LIN {X 0,Y 186.406,Z 165.264,A -85,B 0,C 180,E1 -22320.001,E2 -22320.001} C_VEL
LIN {X 0,Y 185.926,Z 165.321,A -85,B 0,C 180,E1 -22324.336,E2 -22324.336} C_VEL
LIN {X 0,Y 186.028,Z 165.314,A -85,B 0,C 180,E1 -22328.692,E2 -22328.692} C_VEL
LIN {X 0,Y 185.764,Z 165.342,A -85,B 0,C 180,E1 -22333.121,E2 -22333.121} C_VEL
LIN {X 0,Y 185.673,Z 165.354,A -85,B 0,C 180,E1 -22338.867,E2 -22338.867} C_VEL
LIN {X 0,Y 185.576,Z 165.369,A -85,B 0,C 180,E1 -22344.647,E2 -22344.647} C_VEL
LIN {X 0,Y 185.579,Z 165.363,A -85,B 0,C 180,E1 -22349.494,E2 -22349.494} C_VEL
LIN {X 0,Y 185.519,Z 165.374,A -85,B 0,C 180,E1 -22354.629,E2 -22354.629} C_VEL
LIN {X 0,Y 185.544,Z 165.367,A -85,B 0,C 180,E1 -22357.305,E2 -22357.305} C_VEL
LIN {X 0,Y 185.504,Z 165.377,A -85,B 0,C 180,E1 -22360.738,E2 -22360.738} C_VEL
LIN {X 0,Y 185.508,Z 165.375,A -85,B 0,C 180,E1 -22363.962,E2 -22363.962} C_VEL
LIN {X 0,Y 185.485,Z 165.38,A -85,B 0,C 180,E1 -22369.272,E2 -22369.272} C_VEL
LIN {X 0,Y 185.627,Z 165.502,A -85,B 0,C 180,E1 -22372.033,E2 -22372.033} C_VEL
LIN {X 0,Y 187.759,Z 175.884,A -85,B 0,C 180,E1 -22376.802,E2 -22376.802} C_VEL
LIN {X 0,Y 192.861,Z 193.887,A -85,B 0,C 180,E1 -22378.301,E2 -22378.301} C_VEL
LIN {X 0,Y 196.312,Z 235.606,A -85,B 0,C 180,E1 -22380.852,E2 -22380.852} C_VEL
LIN {X 0,Y 194.6,Z 269.087,A -85,B 0,C 180,E1 -22382.53,E2 -22382.53} C_VEL
LIN {X 0,Y 193.581,Z 274.86,A -85,B 0,C 180,E1 -22382.768,E2 -22382.768} C_VEL
LIN {X 0,Y 190.128,Z 284.123,A -85,B 0,C 180,E1 -22383.093,E2 -22383.093} C_VEL
LIN {X 0,Y 186.695,Z 293.281,A -85,B 0,C 180,E1 -22383.622,E2 -22383.622} C_VEL
LIN {X 0,Y 185.665,Z 298.885,A -85,B 0,C 180,E1 -22384.126,E2 -22384.126} C_VEL
LIN {X 0,Y 184.294,Z 310.636,A -85,B 0,C 180,E1 -22385.5,E2 -22385.5} C_VEL
LIN {X 0,Y 182.538,Z 323.588,A -85,B 0,C 180,E1 -22387.526,E2 -22387.526} C_VEL
LIN {X 0,Y 180.854,Z 335.007,A -85,B 0,C 180,E1 -22389.826,E2 -22389.826} C_VEL
LIN {X 0,Y 179.322,Z 344.82,A -85,B 0,C 180,E1 -22392.319,E2 -22392.319} C_VEL
LIN {X 0,Y 178.255,Z 353.885,A -85,B 0,C 180,E1 -22395.152,E2 -22395.152} C_VEL
LIN {X 0,Y 177.417,Z 361.323,A -85,B 0,C 180,E1 -22397.998,E2 -22397.998} C_VEL
LIN {X 0,Y 176.901,Z 368.603,A -85,B 0,C 180,E1 -22401.433,E2 -22401.433} C_VEL
LIN {X 0,Y 176.798,Z 373.802,A -85,B 0,C 180,E1 -22404.512,E2 -22404.512} C_VEL
LIN {X 0,Y 176.75,Z 378.056,A -85,B 0,C 180,E1 -22407.722,E2 -22407.722} C_VEL
LIN {X 0,Y 176.865,Z 380.423,A -85,B 0,C 180,E1 -22410.001,E2 -22410.001} C_VEL
LIN {X 0,Y 176.496,Z 382.213,A -85,B 0,C 180,E1 -22412.283,E2 -22412.283} C_VEL
LIN {X 0,Y 176.293,Z 383.654,A -85,B 0,C 180,E1 -22414.69,E2 -22414.69} C_VEL
LIN {X 0,Y 176.459,Z 385.146,A -85,B 0,C 180,E1 -22419.168,E2 -22419.168} C_VEL
LIN {X 0,Y 177.62,Z 385.137,A -85,B 0,C 180,E1 -22423.734,E2 -22423.734} C_VEL
LIN {X 0,Y 180.063,Z 383.679,A -85,B 0,C 180,E1 -22428.195,E2 -22428.195} C_VEL
LIN {X 0,Y 181.747,Z 382.388,A -85,B 0,C 180,E1 -22430.367,E2 -22430.367} C_VEL
LIN {X 0,Y 185.887,Z 378.597,A -85,B 0,C 180,E1 -22434.576,E2 -22434.576} C_VEL
LIN {X 0,Y 189.751,Z 374.715,A -85,B 0,C 180,E1 -22437.58,E2 -22437.58} C_VEL
LIN {X 0,Y 194.332,Z 369.791,A -85,B 0,C 180,E1 -22440.419,E2 -22440.419} C_VEL
LIN {X 0,Y 200.257,Z 362.613,A -85,B 0,C 180,E1 -22443.556,E2 -22443.556} C_VEL
LIN {X 0,Y 206.088,Z 355.024,A -85,B 0,C 180,E1 -22446.034,E2 -22446.034} C_VEL
LIN {X 0,Y 212.388,Z 345.713,A -85,B 0,C 180,E1 -22448.349,E2 -22448.349} C_VEL
LIN {X 0,Y 219.022,Z 334.32,A -85,B 0,C 180,E1 -22450.526,E2 -22450.526} C_VEL
LIN {X 0,Y 224.449,Z 323.763,A -85,B 0,C 180,E1 -22452.014,E2 -22452.014} C_VEL
LIN {X 0,Y 230.105,Z 310.634,A -85,B 0,C 180,E1 -22453.41,E2 -22453.41} C_VEL
LIN {X 0,Y 234.374,Z 298.405,A -85,B 0,C 180,E1 -22454.352,E2 -22454.352} C_VEL
LIN {X 0,Y 238.04,Z 284.522,A -85,B 0,C 180,E1 -22455.167,E2 -22455.167} C_VEL
LIN {X 0,Y 241.045,Z 267.551,A -85,B 0,C 180,E1 -22455.878,E2 -22455.878} C_VEL
LIN {X 0,Y 243.195,Z 253.201,A -85,B 0,C 180,E1 -22456.447,E2 -22456.447} C_VEL
LIN {X 0,Y 241.769,Z 247.758,A -85,B 0,C 180,E1 -22458.324,E2 -22458.324} C_VEL
LIN {X 0,Y 240.721,Z 244.112,A -85,B 0,C 180,E1 -22459.965,E2 -22459.965} C_VEL
LIN {X 0,Y 239.6,Z 240.401,A -85,B 0,C 180,E1 -22462.093,E2 -22462.093} C_VEL
LIN {X 0,Y 238.583,Z 236.055,A -85,B 0,C 180,E1 -22466.094,E2 -22466.094} C_VEL
LIN {X 0,Y 238.441,Z 235.364,A -85,B 0,C 180,E1 -22467.957,E2 -22467.957} C_VEL
LIN {X 0,Y 238.94,Z 235.62,A -85,B 0,C 180,E1 -22471.095,E2 -22471.095} C_VEL
LIN {X 0,Y 240.37,Z 237.492,A -85,B 0,C 180,E1 -22474.306,E2 -22474.306} C_VEL
LIN {X 0,Y 241.967,Z 240.386,A -85,B 0,C 180,E1 -22476.642,E2 -22476.642} C_VEL
LIN {X 0,Y 243.416,Z 243.368,A -85,B 0,C 180,E1 -22478.363,E2 -22478.363} C_VEL
LIN {X 0,Y 244.149,Z 244.907,A -85,B 0,C 180,E1 -22479.131,E2 -22479.131} C_VEL
LIN {X 0,Y 239.788,Z 272.332,A -85,B 0,C 180,E1 -22480.254,E2 -22480.254} C_VEL
LIN {X 0,Y 236.802,Z 285.281,A -85,B 0,C 180,E1 -22481.057,E2 -22481.057} C_VEL
LIN {X 0,Y 232.723,Z 298.537,A -85,B 0,C 180,E1 -22482.195,E2 -22482.195} C_VEL
LIN {X 0,Y 228.104,Z 310.509,A -85,B 0,C 180,E1 -22483.583,E2 -22483.583} C_VEL
LIN {X 0,Y 223.03,Z 321.088,A -85,B 0,C 180,E1 -22485.141,E2 -22485.141} C_VEL
LIN {X 0,Y 217.786,Z 330.518,A -85,B 0,C 180,E1 -22486.944,E2 -22486.944} C_VEL
LIN {X 0,Y 212.304,Z 339.171,A -85,B 0,C 180,E1 -22489.026,E2 -22489.026} C_VEL
LIN {X 0,Y 207.525,Z 345.733,A -85,B 0,C 180,E1 -22491.023,E2 -22491.023} C_VEL
LIN {X 0,Y 202.253,Z 352.165,A -85,B 0,C 180,E1 -22493.515,E2 -22493.515} C_VEL
LIN {X 0,Y 197.206,Z 357.616,A -85,B 0,C 180,E1 -22496.261,E2 -22496.261} C_VEL
LIN {X 0,Y 192.887,Z 361.653,A -85,B 0,C 180,E1 -22498.955,E2 -22498.955} C_VEL
LIN {X 0,Y 188.616,Z 365.071,A -85,B 0,C 180,E1 -22502.135,E2 -22502.135} C_VEL
LIN {X 0,Y 186.132,Z 366.712,A -85,B 0,C 180,E1 -22504.33,E2 -22504.33} C_VEL
LIN {X 0,Y 183.894,Z 367.917,A -85,B 0,C 180,E1 -22506.583,E2 -22506.583} C_VEL
LIN {X 0,Y 182.006,Z 368.679,A -85,B 0,C 180,E1 -22508.884,E2 -22508.884} C_VEL
LIN {X 0,Y 179.738,Z 368.959,A -85,B 0,C 180,E1 -22512.164,E2 -22512.164} C_VEL
LIN {X 0,Y 177.81,Z 368.208,A -85,B 0,C 180,E1 -22516.061,E2 -22516.061} C_VEL
LIN {X 0,Y 176.957,Z 367.125,A -85,B 0,C 180,E1 -22518.525,E2 -22518.525} C_VEL
LIN {X 0,Y 176.371,Z 365.541,A -85,B 0,C 180,E1 -22521.015,E2 -22521.015} C_VEL
LIN {X 0,Y 176.006,Z 362.223,A -85,B 0,C 180,E1 -22524.788,E2 -22524.788} C_VEL
LIN {X 0,Y 176.163,Z 357.578,A -85,B 0,C 180,E1 -22528.634,E2 -22528.634} C_VEL
LIN {X 0,Y 176.704,Z 351.736,A -85,B 0,C 180,E1 -22532.314,E2 -22532.314} C_VEL
LIN {X 0,Y 177.477,Z 344.811,A -85,B 0,C 180,E1 -22535.738,E2 -22535.738} C_VEL
LIN {X 0,Y 178.528,Z 336.49,A -85,B 0,C 180,E1 -22539.039,E2 -22539.039} C_VEL
LIN {X 0,Y 179.917,Z 326.961,A -85,B 0,C 180,E1 -22542.081,E2 -22542.081} C_VEL
LIN {X 0,Y 181.44,Z 315.862,A -85,B 0,C 180,E1 -22544.909,E2 -22544.909} C_VEL
LIN {X 0,Y 183.087,Z 304.373,A -85,B 0,C 180,E1 -22547.233,E2 -22547.233} C_VEL
LIN {X 0,Y 184.588,Z 292.093,A -85,B 0,C 180,E1 -22549.175,E2 -22549.175} C_VEL
LIN {X 0,Y 185.917,Z 279.648,A -85,B 0,C 180,E1 -22550.683,E2 -22550.683} C_VEL
LIN {X 0,Y 186.97,Z 265.297,A -85,B 0,C 180,E1 -22551.917,E2 -22551.917} C_VEL
LIN {X 0,Y 190.086,Z 210.466,A -85,B 0,C 180,E1 -22554.824,E2 -22554.824} C_VEL
LIN {X 0,Y 190.673,Z 200.076,A -85,B 0,C 180,E1 -22555.357,E2 -22555.357} C_VEL
LIN {X 0,Y 179.22,Z 168.469,A -85,B 0,C 180,E1 -22558.282,E2 -22558.282} C_VEL
LIN {X 0,Y 178.56,Z 166.317,A -85,B 0,C 180,E1 -22558.483,E2 -22558.483} C_VEL
LIN {X 0,Y 178.513,Z 166.249,A -85,B 0,C 180,E1 -22564.337,E2 -22564.337} C_VEL
LIN {X 0,Y 178.521,Z 166.249,A -85,B 0,C 180,E1 -22569.248,E2 -22569.248} C_VEL
LIN {X 0,Y 178.614,Z 166.236,A -85,B 0,C 180,E1 -22571.652,E2 -22571.652} C_VEL
LIN {X 0,Y 178.649,Z 166.226,A -85,B 0,C 180,E1 -22576.346,E2 -22576.346} C_VEL
LIN {X 0,Y 178.958,Z 166.195,A -85,B 0,C 180,E1 -22580.961,E2 -22580.961} C_VEL
LIN {X 0,Y 179.153,Z 166.167,A -85,B 0,C 180,E1 -22587.751,E2 -22587.751} C_VEL
LIN {X 0,Y 179.369,Z 166.141,A -85,B 0,C 180,E1 -22589.999,E2 -22589.999} C_VEL
LIN {X 0,Y 178.872,Z 166.201,A -85,B 0,C 180,E1 -22594.506,E2 -22594.506} C_VEL
LIN {X 0,Y 178.958,Z 166.191,A -85,B 0,C 180,E1 -22599.037,E2 -22599.037} C_VEL
LIN {X 0,Y 178.679,Z 166.226,A -85,B 0,C 180,E1 -22603.65,E2 -22603.65} C_VEL
LIN {X 0,Y 178.62,Z 166.23,A -85,B 0,C 180,E1 -22609.215,E2 -22609.215} C_VEL
LIN {X 0,Y 178.517,Z 166.246,A -85,B 0,C 180,E1 -22615.114,E2 -22615.114} C_VEL
LIN {X 0,Y 178.52,Z 166.246,A -85,B 0,C 180,E1 -22619.993,E2 -22619.993} C_VEL
LIN {X 0,Y 178.482,Z 166.251,A -85,B 0,C 180,E1 -22624.219,E2 -22624.219} C_VEL
LIN {X 0,Y 178.47,Z 166.252,A -85,B 0,C 180,E1 -22629.054,E2 -22629.054} C_VEL
LIN {X 0,Y 178.497,Z 166.25,A -85,B 0,C 180,E1 -22632.015,E2 -22632.015} C_VEL
LIN {X 0,Y 178.514,Z 166.243,A -85,B 0,C 180,E1 -22635.124,E2 -22635.124} C_VEL
LIN {X 0,Y 178.498,Z 166.25,A -85,B 0,C 180,E1 -22638.424,E2 -22638.424} C_VEL
LIN {X 0,Y 178.456,Z 166.254,A -85,B 0,C 180,E1 -22643.792,E2 -22643.792} C_VEL
LIN {X 0,Y 178.489,Z 166.25,A -85,B 0,C 180,E1 -22646.548,E2 -22646.548} C_VEL
LIN {X 0,Y 178.52,Z 166.243,A -85,B 0,C 180,E1 -22650.007,E2 -22650.007} C_VEL
LIN {X 0,Y 178.532,Z 166.246,A -85,B 0,C 180,E1 -22654.876,E2 -22654.876} C_VEL
LIN {X 0,Y 178.621,Z 166.232,A -85,B 0,C 180,E1 -22660.784,E2 -22660.784} C_VEL
LIN {X 0,Y 178.663,Z 166.229,A -85,B 0,C 180,E1 -22664.018,E2 -22664.018} C_VEL
LIN {X 0,Y 178.859,Z 166.204,A -85,B 0,C 180,E1 -22669.211,E2 -22669.211} C_VEL
LIN {X 0,Y 178.923,Z 166.197,A -85,B 0,C 180,E1 -22673.233,E2 -22673.233} C_VEL
LIN {X 0,Y 179.152,Z 166.167,A -85,B 0,C 180,E1 -22677.753,E2 -22677.753} C_VEL
LIN {X 0,Y 179.369,Z 166.141,A -85,B 0,C 180,E1 -22680.001,E2 -22680.001} C_VEL
LIN {X 0,Y 178.875,Z 166.199,A -85,B 0,C 180,E1 -22684.508,E2 -22684.508} C_VEL
LIN {X 0,Y 178.977,Z 166.19,A -85,B 0,C 180,E1 -22689.038,E2 -22689.038} C_VEL
LIN {X 0,Y 178.681,Z 166.224,A -85,B 0,C 180,E1 -22693.651,E2 -22693.651} C_VEL
LIN {X 0,Y 178.621,Z 166.231,A -85,B 0,C 180,E1 -22699.216,E2 -22699.216} C_VEL
LIN {X 0,Y 178.519,Z 166.247,A -85,B 0,C 180,E1 -22705.115,E2 -22705.115} C_VEL
LIN {X 0,Y 178.523,Z 166.244,A -85,B 0,C 180,E1 -22709.995,E2 -22709.995} C_VEL
LIN {X 0,Y 178.496,Z 166.251,A -85,B 0,C 180,E1 -22714.226,E2 -22714.226} C_VEL
LIN {X 0,Y 178.426,Z 166.257,A -85,B 0,C 180,E1 -22719.067,E2 -22719.067} C_VEL
LIN {X 0,Y 178.43,Z 166.26,A -85,B 0,C 180,E1 -22722.037,E2 -22722.037} C_VEL
LIN {X 0,Y 178.422,Z 166.255,A -85,B 0,C 180,E1 -22725.156,E2 -22725.156} C_VEL
LIN {X 0,Y 178.541,Z 166.245,A -85,B 0,C 180,E1 -22731.398,E2 -22731.398} C_VEL
LIN {X 0,Y 178.565,Z 166.455,A -85,B 0,C 180,E1 -22731.709,E2 -22731.709} C_VEL
LIN {X 0,Y 180.436,Z 175.467,A -85,B 0,C 180,E1 -22736.027,E2 -22736.027} C_VEL
LIN {X 0,Y 186.131,Z 195.279,A -85,B 0,C 180,E1 -22737.754,E2 -22737.754} C_VEL
LIN {X 0,Y 189.408,Z 236.226,A -85,B 0,C 180,E1 -22740.353,E2 -22740.353} C_VEL
LIN {X 0,Y 186.805,Z 285.736,A -85,B 0,C 180,E1 -22743.012,E2 -22743.012} C_VEL
LIN {X 0,Y 185.665,Z 298.885,A -85,B 0,C 180,E1 -22744.126,E2 -22744.126} C_VEL
LIN {X 0,Y 184.474,Z 304.383,A -85,B 0,C 180,E1 -22744.679,E2 -22744.679} C_VEL
LIN {X 0,Y 180.587,Z 312.949,A -85,B 0,C 180,E1 -22745.665,E2 -22745.665} C_VEL
LIN {X 0,Y 176.518,Z 321.185,A -85,B 0,C 180,E1 -22746.903,E2 -22746.903} C_VEL
LIN {X 0,Y 175.066,Z 326.174,A -85,B 0,C 180,E1 -22747.839,E2 -22747.839} C_VEL
LIN {X 0,Y 173.279,Z 337.827,A -85,B 0,C 180,E1 -22750.452,E2 -22750.452} C_VEL
LIN {X 0,Y 171.811,Z 348.066,A -85,B 0,C 180,E1 -22753.362,E2 -22753.362} C_VEL
LIN {X 0,Y 170.824,Z 356.454,A -85,B 0,C 180,E1 -22756.317,E2 -22756.317} C_VEL
LIN {X 0,Y 170.017,Z 364.622,A -85,B 0,C 180,E1 -22759.883,E2 -22759.883} C_VEL
LIN {X 0,Y 169.772,Z 371.12,A -85,B 0,C 180,E1 -22763.482,E2 -22763.482} C_VEL
LIN {X 0,Y 169.762,Z 375.361,A -85,B 0,C 180,E1 -22766.441,E2 -22766.441} C_VEL
LIN {X 0,Y 169.846,Z 379.318,A -85,B 0,C 180,E1 -22770.001,E2 -22770.001} C_VEL
LIN {X 0,Y 169.482,Z 381.256,A -85,B 0,C 180,E1 -22772.377,E2 -22772.377} C_VEL
LIN {X 0,Y 169.259,Z 382.734,A -85,B 0,C 180,E1 -22774.764,E2 -22774.764} C_VEL
LIN {X 0,Y 169.462,Z 384.51,A -85,B 0,C 180,E1 -22779.55,E2 -22779.55} C_VEL
LIN {X 0,Y 170.692,Z 384.775,A -85,B 0,C 180,E1 -22784.303,E2 -22784.303} C_VEL
LIN {X 0,Y 173.322,Z 383.535,A -85,B 0,C 180,E1 -22788.93,E2 -22788.93} C_VEL
LIN {X 0,Y 177.157,Z 380.852,A -85,B 0,C 180,E1 -22793.374,E2 -22793.374} C_VEL
LIN {X 0,Y 180.688,Z 377.841,A -85,B 0,C 180,E1 -22796.541,E2 -22796.541} C_VEL
LIN {X 0,Y 185.004,Z 373.829,A -85,B 0,C 180,E1 -22799.595,E2 -22799.595} C_VEL
LIN {X 0,Y 189.968,Z 368.866,A -85,B 0,C 180,E1 -22802.442,E2 -22802.442} C_VEL
LIN {X 0,Y 196.418,Z 361.637,A -85,B 0,C 180,E1 -22805.553,E2 -22805.553} C_VEL
LIN {X 0,Y 202.612,Z 353.914,A -85,B 0,C 180,E1 -22808.003,E2 -22808.003} C_VEL
LIN {X 0,Y 209.266,Z 344.558,A -85,B 0,C 180,E1 -22810.278,E2 -22810.278} C_VEL
LIN {X 0,Y 215.667,Z 334.154,A -85,B 0,C 180,E1 -22812.231,E2 -22812.231} C_VEL
LIN {X 0,Y 221.32,Z 323.646,A -85,B 0,C 180,E1 -22813.684,E2 -22813.684} C_VEL
LIN {X 0,Y 227.164,Z 310.652,A -85,B 0,C 180,E1 -22815.049,E2 -22815.049} C_VEL
LIN {X 0,Y 231.926,Z 297.696,A -85,B 0,C 180,E1 -22816.03,E2 -22816.03} C_VEL
LIN {X 0,Y 235.648,Z 284.377,A -85,B 0,C 180,E1 -22816.782,E2 -22816.782} C_VEL
LIN {X 0,Y 238.358,Z 270.178,A -85,B 0,C 180,E1 -22817.392,E2 -22817.392} C_VEL
LIN {X 0,Y 240.387,Z 256.812,A -85,B 0,C 180,E1 -22817.945,E2 -22817.945} C_VEL
LIN {X 0,Y 239.293,Z 252.159,A -85,B 0,C 180,E1 -22819.748,E2 -22819.748} C_VEL
LIN {X 0,Y 237.982,Z 247.104,A -85,B 0,C 180,E1 -22822.495,E2 -22822.495} C_VEL
LIN {X 0,Y 237.144,Z 242.867,A -85,B 0,C 180,E1 -22826.439,E2 -22826.439} C_VEL
LIN {X 0,Y 237.054,Z 242.37,A -85,B 0,C 180,E1 -22827.747,E2 -22827.747} C_VEL
LIN {X 0,Y 237.498,Z 242.522,A -85,B 0,C 180,E1 -22830.903,E2 -22830.903} C_VEL
LIN {X 0,Y 238.774,Z 244.277,A -85,B 0,C 180,E1 -22833.979,E2 -22833.979} C_VEL
LIN {X 0,Y 240.183,Z 247.037,A -85,B 0,C 180,E1 -22836.219,E2 -22836.219} C_VEL
LIN {X 0,Y 241.264,Z 249.511,A -85,B 0,C 180,E1 -22837.692,E2 -22837.692} C_VEL
LIN {X 0,Y 237.264,Z 273.643,A -85,B 0,C 180,E1 -22838.692,E2 -22838.692} C_VEL
LIN {X 0,Y 234.536,Z 284.996,A -85,B 0,C 180,E1 -22839.382,E2 -22839.382} C_VEL
LIN {X 0,Y 230.604,Z 297.459,A -85,B 0,C 180,E1 -22840.412,E2 -22840.412} C_VEL
LIN {X 0,Y 226.078,Z 308.793,A -85,B 0,C 180,E1 -22841.653,E2 -22841.653} C_VEL
LIN {X 0,Y 220.356,Z 320.659,A -85,B 0,C 180,E1 -22843.318,E2 -22843.318} C_VEL
LIN {X 0,Y 215.439,Z 329.272,A -85,B 0,C 180,E1 -22844.871,E2 -22844.871} C_VEL
LIN {X 0,Y 209.102,Z 338.801,A -85,B 0,C 180,E1 -22847.087,E2 -22847.087} C_VEL
LIN {X 0,Y 202.941,Z 346.839,A -85,B 0,C 180,E1 -22849.524,E2 -22849.524} C_VEL
LIN {X 0,Y 196.777,Z 353.774,A -85,B 0,C 180,E1 -22852.302,E2 -22852.302} C_VEL
LIN {X 0,Y 190.272,Z 360.028,A -85,B 0,C 180,E1 -22855.787,E2 -22855.787} C_VEL
LIN {X 0,Y 185.35,Z 364.002,A -85,B 0,C 180,E1 -22858.913,E2 -22858.913} C_VEL
LIN {X 0,Y 181.062,Z 366.859,A -85,B 0,C 180,E1 -22862.224,E2 -22862.224} C_VEL
LIN {X 0,Y 176.786,Z 368.854,A -85,B 0,C 180,E1 -22866.346,E2 -22866.346} C_VEL
LIN {X 0,Y 174.438,Z 369.415,A -85,B 0,C 180,E1 -22869.273,E2 -22869.273} C_VEL
LIN {X 0,Y 172.542,Z 369.314,A -85,B 0,C 180,E1 -22872.154,E2 -22872.154} C_VEL
LIN {X 0,Y 170.382,Z 367.929,A -85,B 0,C 180,E1 -22876.782,E2 -22876.782} C_VEL
LIN {X 0,Y 169.61,Z 366.506,A -85,B 0,C 180,E1 -22879.358,E2 -22879.358} C_VEL
LIN {X 0,Y 168.948,Z 362.943,A -85,B 0,C 180,E1 -22883.768,E2 -22883.768} C_VEL
LIN {X 0,Y 169.045,Z 357.787,A -85,B 0,C 180,E1 -22888.235,E2 -22888.235} C_VEL
LIN {X 0,Y 169.562,Z 352.162,A -85,B 0,C 180,E1 -22891.9,E2 -22891.9} C_VEL
LIN {X 0,Y 170.262,Z 345.626,A -85,B 0,C 180,E1 -22895.301,E2 -22895.301} C_VEL
LIN {X 0,Y 171.331,Z 337.296,A -85,B 0,C 180,E1 -22898.795,E2 -22898.795} C_VEL
LIN {X 0,Y 172.79,Z 327.298,A -85,B 0,C 180,E1 -22902.152,E2 -22902.152} C_VEL
LIN {X 0,Y 174.246,Z 317.021,A -85,B 0,C 180,E1 -22904.896,E2 -22904.896} C_VEL
LIN {X 0,Y 175.987,Z 305.057,A -85,B 0,C 180,E1 -22907.442,E2 -22907.442} C_VEL
LIN {X 0,Y 177.627,Z 291.82,A -85,B 0,C 180,E1 -22909.608,E2 -22909.608} C_VEL
LIN {X 0,Y 178.903,Z 280.226,A -85,B 0,C 180,E1 -22911.056,E2 -22911.056} C_VEL
LIN {X 0,Y 180.02,Z 265.772,A -85,B 0,C 180,E1 -22912.351,E2 -22912.351} C_VEL
LIN {X 0,Y 183.839,Z 201.675,A -85,B 0,C 180,E1 -22915.862,E2 -22915.862} C_VEL
LIN {X 0,Y 172.963,Z 171.462,A -85,B 0,C 180,E1 -22918.786,E2 -22918.786} C_VEL
LIN {X 0,Y 171.507,Z 167.125,A -85,B 0,C 180,E1 -22919.273,E2 -22919.273} C_VEL
LIN {X 0,Y 171.469,Z 167.127,A -85,B 0,C 180,E1 -22924.382,E2 -22924.382} C_VEL
LIN {X 0,Y 171.546,Z 167.115,A -85,B 0,C 180,E1 -22930.867,E2 -22930.867} C_VEL
LIN {X 0,Y 171.562,Z 167.109,A -85,B 0,C 180,E1 -22935.771,E2 -22935.771} C_VEL
LIN {X 0,Y 171.887,Z 167.074,A -85,B 0,C 180,E1 -22940.586,E2 -22940.586} C_VEL
LIN {X 0,Y 171.821,Z 167.079,A -85,B 0,C 180,E1 -22945.307,E2 -22945.307} C_VEL
LIN {X 0,Y 172.332,Z 167.017,A -85,B 0,C 180,E1 -22949.999,E2 -22949.999} C_VEL
LIN {X 0,Y 171.82,Z 167.08,A -85,B 0,C 180,E1 -22954.692,E2 -22954.692} C_VEL
LIN {X 0,Y 171.887,Z 167.071,A -85,B 0,C 180,E1 -22959.412,E2 -22959.412} C_VEL
LIN {X 0,Y 171.592,Z 167.11,A -85,B 0,C 180,E1 -22964.225,E2 -22964.225} C_VEL
LIN {X 0,Y 171.539,Z 167.111,A -85,B 0,C 180,E1 -22969.559,E2 -22969.559} C_VEL
LIN {X 0,Y 171.456,Z 167.126,A -85,B 0,C 180,E1 -22975.609,E2 -22975.609} C_VEL
LIN {X 0,Y 171.439,Z 167.129,A -85,B 0,C 180,E1 -22980.587,E2 -22980.587} C_VEL
LIN {X 0,Y 171.401,Z 167.13,A -85,B 0,C 180,E1 -22985.032,E2 -22985.032} C_VEL
LIN {X 0,Y 171.424,Z 167.13,A -85,B 0,C 180,E1 -22988.836,E2 -22988.836} C_VEL
LIN {X 0,Y 171.439,Z 167.125,A -85,B 0,C 180,E1 -22994.178,E2 -22994.178} C_VEL
LIN {X 0,Y 171.415,Z 167.132,A -85,B 0,C 180,E1 -22999.006,E2 -22999.006} C_VEL
LIN {X 0,Y 171.434,Z 167.125,A -85,B 0,C 180,E1 -23002.054,E2 -23002.054} C_VEL
LIN {X 0,Y 171.425,Z 167.131,A -85,B 0,C 180,E1 -23007.795,E2 -23007.795} C_VEL
LIN {X 0,Y 171.446,Z 167.123,A -85,B 0,C 180,E1 -23010.535,E2 -23010.535} C_VEL
LIN {X 0,Y 171.455,Z 167.127,A -85,B 0,C 180,E1 -23015.802,E2 -23015.802} C_VEL
LIN {X 0,Y 171.577,Z 167.11,A -85,B 0,C 180,E1 -23020.872,E2 -23020.872} C_VEL
LIN {X 0,Y 171.607,Z 167.106,A -85,B 0,C 180,E1 -23025.776,E2 -23025.776} C_VEL
LIN {X 0,Y 171.886,Z 167.073,A -85,B 0,C 180,E1 -23030.588,E2 -23030.588} C_VEL
LIN {X 0,Y 171.82,Z 167.077,A -85,B 0,C 180,E1 -23035.308,E2 -23035.308} C_VEL
LIN {X 0,Y 172.332,Z 167.017,A -85,B 0,C 180,E1 -23040.001,E2 -23040.001} C_VEL
LIN {X 0,Y 171.824,Z 167.078,A -85,B 0,C 180,E1 -23044.693,E2 -23044.693} C_VEL
LIN {X 0,Y 171.909,Z 167.07,A -85,B 0,C 180,E1 -23049.413,E2 -23049.413} C_VEL
LIN {X 0,Y 171.594,Z 167.108,A -85,B 0,C 180,E1 -23054.227,E2 -23054.227} C_VEL
LIN {X 0,Y 171.541,Z 167.113,A -85,B 0,C 180,E1 -23059.56,E2 -23059.56} C_VEL
LIN {X 0,Y 171.458,Z 167.126,A -85,B 0,C 180,E1 -23065.61,E2 -23065.61} C_VEL
LIN {X 0,Y 171.442,Z 167.128,A -85,B 0,C 180,E1 -23070.588,E2 -23070.588} C_VEL
LIN {X 0,Y 171.407,Z 167.131,A -85,B 0,C 180,E1 -23075.033,E2 -23075.033} C_VEL
LIN {X 0,Y 171.386,Z 167.134,A -85,B 0,C 180,E1 -23078.821,E2 -23078.821} C_VEL
LIN {X 0,Y 171.348,Z 167.137,A -85,B 0,C 180,E1 -23084.21,E2 -23084.21} C_VEL
LIN {X 0,Y 171.36,Z 167.139,A -85,B 0,C 180,E1 -23088.99,E2 -23088.99} C_VEL
LIN {X 0,Y 171.505,Z 167.258,A -85,B 0,C 180,E1 -23091.307,E2 -23091.307} C_VEL
LIN {X 0,Y 173.205,Z 175.333,A -85,B 0,C 180,E1 -23095.253,E2 -23095.253} C_VEL
LIN {X 0,Y 179.382,Z 196.544,A -85,B 0,C 180,E1 -23097.195,E2 -23097.195} C_VEL
LIN {X 0,Y 182.551,Z 235.976,A -85,B 0,C 180,E1 -23099.81,E2 -23099.81} C_VEL
LIN {X 0,Y 179.842,Z 285.434,A -85,B 0,C 180,E1 -23102.588,E2 -23102.588} C_VEL
LIN {X 0,Y 178.562,Z 299.82,A -85,B 0,C 180,E1 -23103.876,E2 -23103.876} C_VEL
LIN {X 0,Y 176.848,Z 313.547,A -85,B 0,C 180,E1 -23105.651,E2 -23105.651} C_VEL
LIN {X 0,Y 175.066,Z 326.174,A -85,B 0,C 180,E1 -23107.839,E2 -23107.839} C_VEL
LIN {X 0,Y 173.649,Z 331.088,A -85,B 0,C 180,E1 -23108.851,E2 -23108.851} C_VEL
LIN {X 0,Y 169.67,Z 338.511,A -85,B 0,C 180,E1 -23110.605,E2 -23110.605} C_VEL
LIN {X 0,Y 165.777,Z 345.442,A -85,B 0,C 180,E1 -23112.623,E2 -23112.623} C_VEL
LIN {X 0,Y 164.512,Z 349.56,A -85,B 0,C 180,E1 -23114.011,E2 -23114.011} C_VEL
LIN {X 0,Y 163.598,Z 357.278,A -85,B 0,C 180,E1 -23116.967,E2 -23116.967} C_VEL
LIN {X 0,Y 162.902,Z 365.144,A -85,B 0,C 180,E1 -23120.69,E2 -23120.69} C_VEL
LIN {X 0,Y 162.751,Z 371.285,A -85,B 0,C 180,E1 -23124.36,E2 -23124.36} C_VEL
LIN {X 0,Y 162.736,Z 375.509,A -85,B 0,C 180,E1 -23127.526,E2 -23127.526} C_VEL
LIN {X 0,Y 162.827,Z 378.147,A -85,B 0,C 180,E1 -23130.001,E2 -23130.001} C_VEL
LIN {X 0,Y 162.464,Z 380.22,A -85,B 0,C 180,E1 -23132.48,E2 -23132.48} C_VEL
LIN {X 0,Y 162.215,Z 381.841,A -85,B 0,C 180,E1 -23134.972,E2 -23134.972} C_VEL
LIN {X 0,Y 162.48,Z 383.827,A -85,B 0,C 180,E1 -23139.964,E2 -23139.964} C_VEL
LIN {X 0,Y 163.79,Z 384.325,A -85,B 0,C 180,E1 -23144.92,E2 -23144.92} C_VEL
LIN {X 0,Y 166.613,Z 383.4,A -85,B 0,C 180,E1 -23149.723,E2 -23149.723} C_VEL
LIN {X 0,Y 170.664,Z 380.97,A -85,B 0,C 180,E1 -23154.319,E2 -23154.319} C_VEL
LIN {X 0,Y 175.808,Z 377.05,A -85,B 0,C 180,E1 -23158.667,E2 -23158.667} C_VEL
LIN {X 0,Y 180.635,Z 373.029,A -85,B 0,C 180,E1 -23161.686,E2 -23161.686} C_VEL
LIN {X 0,Y 185.952,Z 367.991,A -85,B 0,C 180,E1 -23164.537,E2 -23164.537} C_VEL
LIN {X 0,Y 192.861,Z 360.711,A -85,B 0,C 180,E1 -23167.618,E2 -23167.618} C_VEL
LIN {X 0,Y 199.458,Z 352.96,A -85,B 0,C 180,E1 -23170.02,E2 -23170.02} C_VEL
LIN {X 0,Y 206.415,Z 343.513,A -85,B 0,C 180,E1 -23172.257,E2 -23172.257} C_VEL
LIN {X 0,Y 213.165,Z 333.029,A -85,B 0,C 180,E1 -23174.147,E2 -23174.147} C_VEL
LIN {X 0,Y 219.075,Z 322.472,A -85,B 0,C 180,E1 -23175.545,E2 -23175.545} C_VEL
LIN {X 0,Y 225.133,Z 309.43,A -85,B 0,C 180,E1 -23176.862,E2 -23176.862} C_VEL
LIN {X 0,Y 230.17,Z 295.768,A -85,B 0,C 180,E1 -23177.836,E2 -23177.836} C_VEL
LIN {X 0,Y 233.949,Z 282.313,A -85,B 0,C 180,E1 -23178.533,E2 -23178.533} C_VEL
LIN {X 0,Y 237.287,Z 264.378,A -85,B 0,C 180,E1 -23179.267,E2 -23179.267} C_VEL
LIN {X 0,Y 237.841,Z 260.744,A -85,B 0,C 180,E1 -23179.451,E2 -23179.451} C_VEL
LIN {X 0,Y 236.914,Z 256.587,A -85,B 0,C 180,E1 -23181.329,E2 -23181.329} C_VEL
LIN {X 0,Y 236.286,Z 253.567,A -85,B 0,C 180,E1 -23183.137,E2 -23183.137} C_VEL
LIN {X 0,Y 235.717,Z 249.67,A -85,B 0,C 180,E1 -23186.783,E2 -23186.783} C_VEL
LIN {X 0,Y 235.877,Z 249.263,A -85,B 0,C 180,E1 -23189.777,E2 -23189.777} C_VEL
LIN {X 0,Y 236.413,Z 249.978,A -85,B 0,C 180,E1 -23191.893,E2 -23191.893} C_VEL
LIN {X 0,Y 237.25,Z 251.215,A -85,B 0,C 180,E1 -23193.793,E2 -23193.793} C_VEL
LIN {X 0,Y 238.531,Z 253.961,A -85,B 0,C 180,E1 -23195.977,E2 -23195.977} C_VEL
LIN {X 0,Y 238.685,Z 254.361,A -85,B 0,C 180,E1 -23196.218,E2 -23196.218} C_VEL
LIN {X 0,Y 235.05,Z 274.745,A -85,B 0,C 180,E1 -23197.082,E2 -23197.082} C_VEL
LIN {X 0,Y 231.706,Z 287.516,A -85,B 0,C 180,E1 -23197.87,E2 -23197.87} C_VEL
LIN {X 0,Y 227.089,Z 300.871,A -85,B 0,C 180,E1 -23199.004,E2 -23199.004} C_VEL
LIN {X 0,Y 221.997,Z 312.557,A -85,B 0,C 180,E1 -23200.344,E2 -23200.344} C_VEL
LIN {X 0,Y 215.571,Z 324.454,A -85,B 0,C 180,E1 -23202.109,E2 -23202.109} C_VEL
LIN {X 0,Y 209.663,Z 333.719,A -85,B 0,C 180,E1 -23203.945,E2 -23203.945} C_VEL
LIN {X 0,Y 203.601,Z 341.95,A -85,B 0,C 180,E1 -23206.016,E2 -23206.016} C_VEL
LIN {X 0,Y 196.742,Z 349.958,A -85,B 0,C 180,E1 -23208.669,E2 -23208.669} C_VEL
LIN {X 0,Y 190.406,Z 356.321,A -85,B 0,C 180,E1 -23211.509,E2 -23211.509} C_VEL
LIN {X 0,Y 184.908,Z 361.098,A -85,B 0,C 180,E1 -23214.382,E2 -23214.382} C_VEL
LIN {X 0,Y 179.36,Z 365.085,A -85,B 0,C 180,E1 -23217.754,E2 -23217.754} C_VEL
LIN {X 0,Y 175.707,Z 367.255,A -85,B 0,C 180,E1 -23220.418,E2 -23220.418} C_VEL
LIN {X 0,Y 170.949,Z 369.33,A -85,B 0,C 180,E1 -23224.716,E2 -23224.716} C_VEL
LIN {X 0,Y 168.739,Z 369.831,A -85,B 0,C 180,E1 -23227.177,E2 -23227.177} C_VEL
LIN {X 0,Y 166.853,Z 369.909,A -85,B 0,C 180,E1 -23229.699,E2 -23229.699} C_VEL
LIN {X 0,Y 165.258,Z 369.533,A -85,B 0,C 180,E1 -23232.276,E2 -23232.276} C_VEL
LIN {X 0,Y 163.964,Z 368.681,A -85,B 0,C 180,E1 -23234.902,E2 -23234.902} C_VEL
LIN {X 0,Y 162.789,Z 367.003,A -85,B 0,C 180,E1 -23238.23,E2 -23238.23} C_VEL
LIN {X 0,Y 161.9,Z 363.3,A -85,B 0,C 180,E1 -23242.996,E2 -23242.996} C_VEL
LIN {X 0,Y 161.869,Z 358.822,A -85,B 0,C 180,E1 -23247.121,E2 -23247.121} C_VEL
LIN {X 0,Y 162.373,Z 352.857,A -85,B 0,C 180,E1 -23251.291,E2 -23251.291} C_VEL
LIN {X 0,Y 163.086,Z 345.974,A -85,B 0,C 180,E1 -23255.035,E2 -23255.035} C_VEL
LIN {X 0,Y 164.067,Z 338.341,A -85,B 0,C 180,E1 -23258.397,E2 -23258.397} C_VEL
LIN {X 0,Y 165.519,Z 328.293,A -85,B 0,C 180,E1 -23261.969,E2 -23261.969} C_VEL
LIN {X 0,Y 166.991,Z 318.421,A -85,B 0,C 180,E1 -23264.769,E2 -23264.769} C_VEL
LIN {X 0,Y 168.594,Z 307.454,A -85,B 0,C 180,E1 -23267.282,E2 -23267.282} C_VEL
LIN {X 0,Y 170.187,Z 295.8,A -85,B 0,C 180,E1 -23269.406,E2 -23269.406} C_VEL
LIN {X 0,Y 171.826,Z 281.69,A -85,B 0,C 180,E1 -23271.342,E2 -23271.342} C_VEL
LIN {X 0,Y 172.926,Z 268.147,A -85,B 0,C 180,E1 -23272.674,E2 -23272.674} C_VEL
LIN {X 0,Y 174.232,Z 246.373,A -85,B 0,C 180,E1 -23274.022,E2 -23274.022} C_VEL
LIN {X 0,Y 176.918,Z 202.961,A -85,B 0,C 180,E1 -23276.434,E2 -23276.434} C_VEL
LIN {X 0,Y 166.672,Z 174.336,A -85,B 0,C 180,E1 -23279.307,E2 -23279.307} C_VEL
LIN {X 0,Y 164.437,Z 168.005,A -85,B 0,C 180,E1 -23280.031,E2 -23280.031} C_VEL
LIN {X 0,Y 164.416,Z 168.006,A -85,B 0,C 180,E1 -23284.693,E2 -23284.693} C_VEL
LIN {X 0,Y 164.443,Z 167.999,A -85,B 0,C 180,E1 -23290.089,E2 -23290.089} C_VEL
LIN {X 0,Y 164.489,Z 167.993,A -85,B 0,C 180,E1 -23295.145,E2 -23295.145} C_VEL
LIN {X 0,Y 164.801,Z 167.956,A -85,B 0,C 180,E1 -23300.177,E2 -23300.177} C_VEL
LIN {X 0,Y 164.85,Z 167.95,A -85,B 0,C 180,E1 -23302.651,E2 -23302.651} C_VEL
LIN {X 0,Y 165.049,Z 167.925,A -85,B 0,C 180,E1 -23307.559,E2 -23307.559} C_VEL
LIN {X 0,Y 165.294,Z 167.894,A -85,B 0,C 180,E1 -23309.999,E2 -23309.999} C_VEL
LIN {X 0,Y 164.77,Z 167.96,A -85,B 0,C 180,E1 -23314.893,E2 -23314.893} C_VEL
LIN {X 0,Y 164.849,Z 167.95,A -85,B 0,C 180,E1 -23317.347,E2 -23317.347} C_VEL
LIN {X 0,Y 164.752,Z 167.957,A -85,B 0,C 180,E1 -23321.151,E2 -23321.151} C_VEL
LIN {X 0,Y 164.483,Z 167.994,A -85,B 0,C 180,E1 -23327.402,E2 -23327.402} C_VEL
LIN {X 0,Y 164.47,Z 167.993,A -85,B 0,C 180,E1 -23329.989,E2 -23329.989} C_VEL
LIN {X 0,Y 164.383,Z 168.007,A -85,B 0,C 180,E1 -23336.128,E2 -23336.128} C_VEL
LIN {X 0,Y 164.373,Z 168.009,A -85,B 0,C 180,E1 -23341.228,E2 -23341.228} C_VEL
LIN {X 0,Y 164.345,Z 168.009,A -85,B 0,C 180,E1 -23346.775,E2 -23346.775} C_VEL
LIN {X 0,Y 164.366,Z 168.012,A -85,B 0,C 180,E1 -23349.893,E2 -23349.893} C_VEL
LIN {X 0,Y 164.376,Z 168.007,A -85,B 0,C 180,E1 -23353.379,E2 -23353.379} C_VEL
LIN {X 0,Y 164.38,Z 168.007,A -85,B 0,C 180,E1 -23356.839,E2 -23356.839} C_VEL
LIN {X 0,Y 164.367,Z 168.009,A -85,B 0,C 180,E1 -23360.32,E2 -23360.32} C_VEL
LIN {X 0,Y 164.342,Z 168.011,A -85,B 0,C 180,E1 -23364.342,E2 -23364.342} C_VEL
LIN {X 0,Y 164.403,Z 168.005,A -85,B 0,C 180,E1 -23369.138,E2 -23369.138} C_VEL
LIN {X 0,Y 164.414,Z 168.004,A -85,B 0,C 180,E1 -23374.695,E2 -23374.695} C_VEL
LIN {X 0,Y 164.482,Z 167.992,A -85,B 0,C 180,E1 -23380.052,E2 -23380.052} C_VEL
LIN {X 0,Y 164.551,Z 167.987,A -85,B 0,C 180,E1 -23385.153,E2 -23385.153} C_VEL
LIN {X 0,Y 164.806,Z 167.954,A -85,B 0,C 180,E1 -23390.18,E2 -23390.18} C_VEL
LIN {X 0,Y 164.849,Z 167.951,A -85,B 0,C 180,E1 -23392.653,E2 -23392.653} C_VEL
LIN {X 0,Y 165.048,Z 167.924,A -85,B 0,C 180,E1 -23397.56,E2 -23397.56} C_VEL
LIN {X 0,Y 165.294,Z 167.894,A -85,B 0,C 180,E1 -23400.001,E2 -23400.001} C_VEL
LIN {X 0,Y 164.775,Z 167.957,A -85,B 0,C 180,E1 -23404.894,E2 -23404.894} C_VEL
LIN {X 0,Y 164.861,Z 167.948,A -85,B 0,C 180,E1 -23407.349,E2 -23407.349} C_VEL
LIN {X 0,Y 164.779,Z 167.955,A -85,B 0,C 180,E1 -23411.199,E2 -23411.199} C_VEL
LIN {X 0,Y 164.484,Z 167.995,A -85,B 0,C 180,E1 -23417.404,E2 -23417.404} C_VEL
LIN {X 0,Y 164.472,Z 167.995,A -85,B 0,C 180,E1 -23419.99,E2 -23419.99} C_VEL
LIN {X 0,Y 164.385,Z 168.009,A -85,B 0,C 180,E1 -23426.13,E2 -23426.13} C_VEL
LIN {X 0,Y 164.376,Z 168.007,A -85,B 0,C 180,E1 -23431.23,E2 -23431.23} C_VEL
LIN {X 0,Y 164.314,Z 168.011,A -85,B 0,C 180,E1 -23436.785,E2 -23436.785} C_VEL
LIN {X 0,Y 164.306,Z 168.018,A -85,B 0,C 180,E1 -23439.913,E2 -23439.913} C_VEL
LIN {X 0,Y 164.307,Z 168.017,A -85,B 0,C 180,E1 -23443.353,E2 -23443.353} C_VEL
LIN {X 0,Y 164.293,Z 168.019,A -85,B 0,C 180,E1 -23446.81,E2 -23446.81} C_VEL
LIN {X 0,Y 164.417,Z 168.091,A -85,B 0,C 180,E1 -23450.914,E2 -23450.914} C_VEL
LIN {X 0,Y 165.865,Z 174.967,A -85,B 0,C 180,E1 -23454.393,E2 -23454.393} C_VEL
LIN {X 0,Y 172.649,Z 198.493,A -85,B 0,C 180,E1 -23456.648,E2 -23456.648} C_VEL
LIN {X 0,Y 175.596,Z 237.151,A -85,B 0,C 180,E1 -23459.317,E2 -23459.317} C_VEL
LIN {X 0,Y 172.893,Z 285.135,A -85,B 0,C 180,E1 -23462.131,E2 -23462.131} C_VEL
LIN {X 0,Y 171.649,Z 298.818,A -85,B 0,C 180,E1 -23463.397,E2 -23463.397} C_VEL
LIN {X 0,Y 170.155,Z 310.846,A -85,B 0,C 180,E1 -23464.954,E2 -23464.954} C_VEL
LIN {X 0,Y 168.33,Z 323.897,A -85,B 0,C 180,E1 -23467.203,E2 -23467.203} C_VEL
LIN {X 0,Y 166.628,Z 334.813,A -85,B 0,C 180,E1 -23469.638,E2 -23469.638} C_VEL
LIN {X 0,Y 164.996,Z 345.477,A -85,B 0,C 180,E1 -23472.654,E2 -23472.654} C_VEL
LIN {X 0,Y 164.512,Z 349.56,A -85,B 0,C 180,E1 -23474.011,E2 -23474.011} C_VEL
LIN {X 0,Y 163.314,Z 353.537,A -85,B 0,C 180,E1 -23475.48,E2 -23475.48} C_VEL
LIN {X 0,Y 159.81,Z 359.338,A -85,B 0,C 180,E1 -23478.049,E2 -23478.049} C_VEL
LIN {X 0,Y 156.552,Z 364.541,A -85,B 0,C 180,E1 -23480.895,E2 -23480.895} C_VEL
LIN {X 0,Y 155.762,Z 367.587,A -85,B 0,C 180,E1 -23482.746,E2 -23482.746} C_VEL
LIN {X 0,Y 155.736,Z 372.548,A -85,B 0,C 180,E1 -23486.12,E2 -23486.12} C_VEL
LIN {X 0,Y 155.829,Z 376.95,A -85,B 0,C 180,E1 -23490.001,E2 -23490.001} C_VEL
LIN {X 0,Y 155.462,Z 379.11,A -85,B 0,C 180,E1 -23492.592,E2 -23492.592} C_VEL
LIN {X 0,Y 155.232,Z 382.163,A -85,B 0,C 180,E1 -23497.807,E2 -23497.807} C_VEL
LIN {X 0,Y 156.06,Z 383.677,A -85,B 0,C 180,E1 -23503.014,E2 -23503.014} C_VEL
LIN {X 0,Y 158.233,Z 383.688,A -85,B 0,C 180,E1 -23508.115,E2 -23508.115} C_VEL
LIN {X 0,Y 161.888,Z 382.292,A -85,B 0,C 180,E1 -23513,E2 -23513} C_VEL
LIN {X 0,Y 166.77,Z 379.474,A -85,B 0,C 180,E1 -23517.618,E2 -23517.618} C_VEL
LIN {X 0,Y 171.231,Z 376.335,A -85,B 0,C 180,E1 -23520.868,E2 -23520.868} C_VEL
LIN {X 0,Y 176.452,Z 372.242,A -85,B 0,C 180,E1 -23523.892,E2 -23523.892} C_VEL
LIN {X 0,Y 182.177,Z 367.208,A -85,B 0,C 180,E1 -23526.725,E2 -23526.725} C_VEL
LIN {X 0,Y 188.514,Z 361.009,A -85,B 0,C 180,E1 -23529.33,E2 -23529.33} C_VEL
LIN {X 0,Y 195.368,Z 353.444,A -85,B 0,C 180,E1 -23531.722,E2 -23531.722} C_VEL
LIN {X 0,Y 202.624,Z 344.35,A -85,B 0,C 180,E1 -23533.924,E2 -23533.924} C_VEL
LIN {X 0,Y 209.611,Z 334.173,A -85,B 0,C 180,E1 -23535.782,E2 -23535.782} C_VEL
LIN {X 0,Y 215.705,Z 323.971,A -85,B 0,C 180,E1 -23537.147,E2 -23537.147} C_VEL
LIN {X 0,Y 221.958,Z 311.49,A -85,B 0,C 180,E1 -23538.423,E2 -23538.423} C_VEL
LIN {X 0,Y 227.502,Z 297.862,A -85,B 0,C 180,E1 -23539.426,E2 -23539.426} C_VEL
LIN {X 0,Y 231.76,Z 283.911,A -85,B 0,C 180,E1 -23540.167,E2 -23540.167} C_VEL
LIN {X 0,Y 234.746,Z 269.838,A -85,B 0,C 180,E1 -23540.737,E2 -23540.737} C_VEL
LIN {X 0,Y 235.537,Z 265.092,A -85,B 0,C 180,E1 -23540.929,E2 -23540.929} C_VEL
LIN {X 0,Y 234.991,Z 262.132,A -85,B 0,C 180,E1 -23542.424,E2 -23542.424} C_VEL
LIN {X 0,Y 234.626,Z 259.908,A -85,B 0,C 180,E1 -23543.821,E2 -23543.821} C_VEL
LIN {X 0,Y 234.296,Z 256.483,A -85,B 0,C 180,E1 -23547.13,E2 -23547.13} C_VEL
LIN {X 0,Y 234.665,Z 256.382,A -85,B 0,C 180,E1 -23550.723,E2 -23550.723} C_VEL
LIN {X 0,Y 235.666,Z 258.034,A -85,B 0,C 180,E1 -23553.466,E2 -23553.466} C_VEL
LIN {X 0,Y 236.277,Z 259.363,A -85,B 0,C 180,E1 -23554.724,E2 -23554.724} C_VEL
LIN {X 0,Y 232.966,Z 276.774,A -85,B 0,C 180,E1 -23555.471,E2 -23555.471} C_VEL
LIN {X 0,Y 229.247,Z 289.901,A -85,B 0,C 180,E1 -23556.302,E2 -23556.302} C_VEL
LIN {X 0,Y 225.023,Z 301.328,A -85,B 0,C 180,E1 -23557.262,E2 -23557.262} C_VEL
LIN {X 0,Y 220.218,Z 311.924,A -85,B 0,C 180,E1 -23558.44,E2 -23558.44} C_VEL
LIN {X 0,Y 213.855,Z 323.466,A -85,B 0,C 180,E1 -23560.064,E2 -23560.064} C_VEL
LIN {X 0,Y 208.175,Z 332.222,A -85,B 0,C 180,E1 -23561.666,E2 -23561.666} C_VEL
LIN {X 0,Y 201.39,Z 341.199,A -85,B 0,C 180,E1 -23563.788,E2 -23563.788} C_VEL
LIN {X 0,Y 194.063,Z 349.43,A -85,B 0,C 180,E1 -23566.383,E2 -23566.383} C_VEL
LIN {X 0,Y 187.251,Z 356.02,A -85,B 0,C 180,E1 -23569.183,E2 -23569.183} C_VEL
LIN {X 0,Y 180.928,Z 361.19,A -85,B 0,C 180,E1 -23572.185,E2 -23572.185} C_VEL
LIN {X 0,Y 175.239,Z 365.123,A -85,B 0,C 180,E1 -23575.398,E2 -23575.398} C_VEL
LIN {X 0,Y 171.771,Z 367.098,A -85,B 0,C 180,E1 -23577.654,E2 -23577.654} C_VEL
LIN {X 0,Y 168.654,Z 368.593,A -85,B 0,C 180,E1 -23579.999,E2 -23579.999} C_VEL
LIN {X 0,Y 165.846,Z 369.654,A -85,B 0,C 180,E1 -23582.428,E2 -23582.428} C_VEL
LIN {X 0,Y 162.493,Z 370.353,A -85,B 0,C 180,E1 -23585.852,E2 -23585.852} C_VEL
LIN {X 0,Y 159.265,Z 370.138,A -85,B 0,C 180,E1 -23590.166,E2 -23590.166} C_VEL
LIN {X 0,Y 157.744,Z 369.417,A -85,B 0,C 180,E1 -23592.871,E2 -23592.871} C_VEL
LIN {X 0,Y 156.495,Z 368.221,A -85,B 0,C 180,E1 -23595.631,E2 -23595.631} C_VEL
LIN {X 0,Y 155.279,Z 365.564,A -85,B 0,C 180,E1 -23599.841,E2 -23599.841} C_VEL
LIN {X 0,Y 154.761,Z 361.107,A -85,B 0,C 180,E1 -23604.735,E2 -23604.735} C_VEL
LIN {X 0,Y 154.99,Z 355.593,A -85,B 0,C 180,E1 -23609.173,E2 -23609.173} C_VEL
LIN {X 0,Y 155.714,Z 348.515,A -85,B 0,C 180,E1 -23613.565,E2 -23613.565} C_VEL
LIN {X 0,Y 156.563,Z 341.29,A -85,B 0,C 180,E1 -23617.138,E2 -23617.138} C_VEL
LIN {X 0,Y 157.818,Z 332.086,A -85,B 0,C 180,E1 -23620.794,E2 -23620.794} C_VEL
LIN {X 0,Y 159.374,Z 322.046,A -85,B 0,C 180,E1 -23623.989,E2 -23623.989} C_VEL
LIN {X 0,Y 161.007,Z 311.339,A -85,B 0,C 180,E1 -23626.738,E2 -23626.738} C_VEL
LIN {X 0,Y 162.814,Z 298.519,A -85,B 0,C 180,E1 -23629.309,E2 -23629.309} C_VEL
LIN {X 0,Y 164.383,Z 285.683,A -85,B 0,C 180,E1 -23631.283,E2 -23631.283} C_VEL
LIN {X 0,Y 165.726,Z 271.536,A -85,B 0,C 180,E1 -23632.855,E2 -23632.855} C_VEL
LIN {X 0,Y 166.738,Z 257.222,A -85,B 0,C 180,E1 -23633.91,E2 -23633.91} C_VEL
LIN {X 0,Y 170.024,Z 204.294,A -85,B 0,C 180,E1 -23637.019,E2 -23637.019} C_VEL
LIN {X 0,Y 160.051,Z 176.351,A -85,B 0,C 180,E1 -23639.942,E2 -23639.942} C_VEL
LIN {X 0,Y 157.348,Z 168.889,A -85,B 0,C 180,E1 -23640.847,E2 -23640.847} C_VEL
LIN {X 0,Y 157.31,Z 168.891,A -85,B 0,C 180,E1 -23646.29,E2 -23646.29} C_VEL
LIN {X 0,Y 157.378,Z 168.881,A -85,B 0,C 180,E1 -23651.783,E2 -23651.783} C_VEL
LIN {X 0,Y 157.531,Z 168.858,A -85,B 0,C 180,E1 -23657.11,E2 -23657.11} C_VEL
LIN {X 0,Y 157.725,Z 168.837,A -85,B 0,C 180,E1 -23659.732,E2 -23659.732} C_VEL
LIN {X 0,Y 157.807,Z 168.827,A -85,B 0,C 180,E1 -23662.321,E2 -23662.321} C_VEL
LIN {X 0,Y 158.257,Z 168.771,A -85,B 0,C 180,E1 -23669.999,E2 -23669.999} C_VEL
LIN {X 0,Y 157.807,Z 168.827,A -85,B 0,C 180,E1 -23677.677,E2 -23677.677} C_VEL
LIN {X 0,Y 157.681,Z 168.838,A -85,B 0,C 180,E1 -23681.32,E2 -23681.32} C_VEL
LIN {X 0,Y 157.46,Z 168.87,A -85,B 0,C 180,E1 -23685.532,E2 -23685.532} C_VEL
LIN {X 0,Y 157.365,Z 168.881,A -85,B 0,C 180,E1 -23690.932,E2 -23690.932} C_VEL
LIN {X 0,Y 157.306,Z 168.886,A -85,B 0,C 180,E1 -23696.68,E2 -23696.68} C_VEL
LIN {X 0,Y 157.275,Z 168.894,A -85,B 0,C 180,E1 -23702.426,E2 -23702.426} C_VEL
LIN {X 0,Y 157.319,Z 168.885,A -85,B 0,C 180,E1 -23706.476,E2 -23706.476} C_VEL
LIN {X 0,Y 157.284,Z 168.892,A -85,B 0,C 180,E1 -23712.085,E2 -23712.085} C_VEL
LIN {X 0,Y 157.299,Z 168.887,A -85,B 0,C 180,E1 -23715.631,E2 -23715.631} C_VEL
LIN {X 0,Y 157.284,Z 168.891,A -85,B 0,C 180,E1 -23721.277,E2 -23721.277} C_VEL
LIN {X 0,Y 157.289,Z 168.89,A -85,B 0,C 180,E1 -23724.49,E2 -23724.49} C_VEL
LIN {X 0,Y 157.299,Z 168.89,A -85,B 0,C 180,E1 -23728.091,E2 -23728.091} C_VEL
LIN {X 0,Y 157.319,Z 168.888,A -85,B 0,C 180,E1 -23733.467,E2 -23733.467} C_VEL
LIN {X 0,Y 157.391,Z 168.876,A -85,B 0,C 180,E1 -23739.668,E2 -23739.668} C_VEL
LIN {X 0,Y 157.476,Z 168.868,A -85,B 0,C 180,E1 -23744.469,E2 -23744.469} C_VEL
LIN {X 0,Y 157.733,Z 168.836,A -85,B 0,C 180,E1 -23749.735,E2 -23749.735} C_VEL
LIN {X 0,Y 157.807,Z 168.827,A -85,B 0,C 180,E1 -23752.323,E2 -23752.323} C_VEL
LIN {X 0,Y 158.256,Z 168.771,A -85,B 0,C 180,E1 -23760.001,E2 -23760.001} C_VEL
LIN {X 0,Y 157.823,Z 168.825,A -85,B 0,C 180,E1 -23767.678,E2 -23767.678} C_VEL
LIN {X 0,Y 157.704,Z 168.836,A -85,B 0,C 180,E1 -23771.362,E2 -23771.362} C_VEL
LIN {X 0,Y 157.461,Z 168.87,A -85,B 0,C 180,E1 -23775.534,E2 -23775.534} C_VEL
LIN {X 0,Y 157.366,Z 168.878,A -85,B 0,C 180,E1 -23780.934,E2 -23780.934} C_VEL
LIN {X 0,Y 157.309,Z 168.888,A -85,B 0,C 180,E1 -23786.682,E2 -23786.682} C_VEL
LIN {X 0,Y 157.278,Z 168.894,A -85,B 0,C 180,E1 -23792.428,E2 -23792.428} C_VEL
LIN {X 0,Y 157.284,Z 168.888,A -85,B 0,C 180,E1 -23796.459,E2 -23796.459} C_VEL
LIN {X 0,Y 157.215,Z 168.902,A -85,B 0,C 180,E1 -23802.111,E2 -23802.111} C_VEL
LIN {X 0,Y 157.229,Z 168.902,A -85,B 0,C 180,E1 -23807.897,E2 -23807.897} C_VEL
LIN {X 0,Y 157.332,Z 168.919,A -85,B 0,C 180,E1 -23810.508,E2 -23810.508} C_VEL
LIN {X 0,Y 158.475,Z 174.235,A -85,B 0,C 180,E1 -23813.435,E2 -23813.435} C_VEL
LIN {X 0,Y 165.869,Z 199.437,A -85,B 0,C 180,E1 -23816.006,E2 -23816.006} C_VEL
LIN {X 0,Y 168.724,Z 237.207,A -85,B 0,C 180,E1 -23818.724,E2 -23818.724} C_VEL
LIN {X 0,Y 165.963,Z 284.58,A -85,B 0,C 180,E1 -23821.637,E2 -23821.637} C_VEL
LIN {X 0,Y 164.63,Z 298.87,A -85,B 0,C 180,E1 -23823.028,E2 -23823.028} C_VEL
LIN {X 0,Y 162.991,Z 311.738,A -85,B 0,C 180,E1 -23824.818,E2 -23824.818} C_VEL
LIN {X 0,Y 161.328,Z 323.252,A -85,B 0,C 180,E1 -23826.918,E2 -23826.918} C_VEL
LIN {X 0,Y 159.624,Z 333.89,A -85,B 0,C 180,E1 -23829.377,E2 -23829.377} C_VEL
LIN {X 0,Y 157.972,Z 344.642,A -85,B 0,C 180,E1 -23832.525,E2 -23832.525} C_VEL
LIN {X 0,Y 156.896,Z 353.484,A -85,B 0,C 180,E1 -23835.738,E2 -23835.738} C_VEL
LIN {X 0,Y 156.118,Z 360.737,A -85,B 0,C 180,E1 -23838.971,E2 -23838.971} C_VEL
LIN {X 0,Y 155.762,Z 367.587,A -85,B 0,C 180,E1 -23842.746,E2 -23842.746} C_VEL
LIN {X 0,Y 155.038,Z 370.395,A -85,B 0,C 180,E1 -23844.647,E2 -23844.647} C_VEL
LIN {X 0,Y 153.45,Z 372.74,A -85,B 0,C 180,E1 -23846.592,E2 -23846.592} C_VEL
LIN {X 0,Y 149.687,Z 376.466,A -85,B 0,C 180,E1 -23850.698,E2 -23850.698} C_VEL
LIN {X 0,Y 148.349,Z 378.59,A -85,B 0,C 180,E1 -23853.644,E2 -23853.644} C_VEL
LIN {X 0,Y 148.246,Z 381.258,A -85,B 0,C 180,E1 -23858.177,E2 -23858.177} C_VEL
LIN {X 0,Y 149.147,Z 382.983,A -85,B 0,C 180,E1 -23863.628,E2 -23863.628} C_VEL
LIN {X 0,Y 151.5,Z 383.31,A -85,B 0,C 180,E1 -23868.95,E2 -23868.95} C_VEL
LIN {X 0,Y 155.366,Z 382.196,A -85,B 0,C 180,E1 -23874.025,E2 -23874.025} C_VEL
LIN {X 0,Y 160.81,Z 379.467,A -85,B 0,C 180,E1 -23879.062,E2 -23879.062} C_VEL
LIN {X 0,Y 166.92,Z 375.653,A -85,B 0,C 180,E1 -23883.186,E2 -23883.186} C_VEL
LIN {X 0,Y 172.553,Z 371.567,A -85,B 0,C 180,E1 -23886.199,E2 -23886.199} C_VEL
LIN {X 0,Y 178.694,Z 366.473,A -85,B 0,C 180,E1 -23888.998,E2 -23888.998} C_VEL
LIN {X 0,Y 186.646,Z 359.114,A -85,B 0,C 180,E1 -23891.942,E2 -23891.942} C_VEL
LIN {X 0,Y 193.945,Z 351.315,A -85,B 0,C 180,E1 -23894.233,E2 -23894.233} C_VEL
LIN {X 0,Y 201.588,Z 341.839,A -85,B 0,C 180,E1 -23896.338,E2 -23896.338} C_VEL
LIN {X 0,Y 208.299,Z 332.36,A -85,B 0,C 180,E1 -23897.927,E2 -23897.927} C_VEL
LIN {X 0,Y 215.36,Z 320.675,A -85,B 0,C 180,E1 -23899.354,E2 -23899.354} C_VEL
LIN {X 0,Y 221.67,Z 307.998,A -85,B 0,C 180,E1 -23900.5,E2 -23900.5} C_VEL
LIN {X 0,Y 226.844,Z 294.816,A -85,B 0,C 180,E1 -23901.359,E2 -23901.359} C_VEL
LIN {X 0,Y 231.032,Z 280.948,A -85,B 0,C 180,E1 -23902.023,E2 -23902.023} C_VEL
LIN {X 0,Y 233.458,Z 269.5,A -85,B 0,C 180,E1 -23902.494,E2 -23902.494} C_VEL
LIN {X 0,Y 233.075,Z 266.779,A -85,B 0,C 180,E1 -23904.146,E2 -23904.146} C_VEL
LIN {X 0,Y 232.879,Z 263.324,A -85,B 0,C 180,E1 -23907.486,E2 -23907.486} C_VEL
LIN {X 0,Y 233.287,Z 263.46,A -85,B 0,C 180,E1 -23910.887,E2 -23910.887} C_VEL
LIN {X 0,Y 234.113,Z 264.899,A -85,B 0,C 180,E1 -23913.196,E2 -23913.196} C_VEL
LIN {X 0,Y 231.022,Z 279.237,A -85,B 0,C 180,E1 -23913.862,E2 -23913.862} C_VEL
LIN {X 0,Y 227.345,Z 291.225,A -85,B 0,C 180,E1 -23914.625,E2 -23914.625} C_VEL
LIN {X 0,Y 222.182,Z 304.284,A -85,B 0,C 180,E1 -23915.718,E2 -23915.718} C_VEL
LIN {X 0,Y 216.381,Z 315.966,A -85,B 0,C 180,E1 -23917.06,E2 -23917.06} C_VEL
LIN {X 0,Y 209.89,Z 326.673,A -85,B 0,C 180,E1 -23918.645,E2 -23918.645} C_VEL
LIN {X 0,Y 202.436,Z 336.931,A -85,B 0,C 180,E1 -23920.672,E2 -23920.672} C_VEL
LIN {X 0,Y 195.626,Z 344.986,A -85,B 0,C 180,E1 -23922.758,E2 -23922.758} C_VEL
LIN {X 0,Y 188.17,Z 352.448,A -85,B 0,C 180,E1 -23925.341,E2 -23925.341} C_VEL
LIN {X 0,Y 179.897,Z 359.446,A -85,B 0,C 180,E1 -23928.735,E2 -23928.735} C_VEL
LIN {X 0,Y 173.503,Z 363.935,A -85,B 0,C 180,E1 -23931.849,E2 -23931.849} C_VEL
LIN {X 0,Y 167.657,Z 367.242,A -85,B 0,C 180,E1 -23935.19,E2 -23935.19} C_VEL
LIN {X 0,Y 161.653,Z 369.753,A -85,B 0,C 180,E1 -23939.474,E2 -23939.474} C_VEL
LIN {X 0,Y 158.214,Z 370.664,A -85,B 0,C 180,E1 -23942.545,E2 -23942.545} C_VEL
LIN {X 0,Y 155.349,Z 370.896,A -85,B 0,C 180,E1 -23945.559,E2 -23945.559} C_VEL
LIN {X 0,Y 151.676,Z 370.099,A -85,B 0,C 180,E1 -23950.68,E2 -23950.68} C_VEL
LIN {X 0,Y 150.229,Z 369.029,A -85,B 0,C 180,E1 -23953.526,E2 -23953.526} C_VEL
LIN {X 0,Y 148.407,Z 365.957,A -85,B 0,C 180,E1 -23958.713,E2 -23958.713} C_VEL
LIN {X 0,Y 147.703,Z 361.547,A -85,B 0,C 180,E1 -23963.809,E2 -23963.809} C_VEL
LIN {X 0,Y 147.843,Z 356.14,A -85,B 0,C 180,E1 -23968.382,E2 -23968.382} C_VEL
LIN {X 0,Y 148.515,Z 349.117,A -85,B 0,C 180,E1 -23972.969,E2 -23972.969} C_VEL
LIN {X 0,Y 149.369,Z 341.592,A -85,B 0,C 180,E1 -23976.881,E2 -23976.881} C_VEL
LIN {X 0,Y 150.68,Z 332.274,A -85,B 0,C 180,E1 -23980.766,E2 -23980.766} C_VEL
LIN {X 0,Y 152.335,Z 321.807,A -85,B 0,C 180,E1 -23984.249,E2 -23984.249} C_VEL
LIN {X 0,Y 153.896,Z 311.751,A -85,B 0,C 180,E1 -23986.942,E2 -23986.942} C_VEL
LIN {X 0,Y 155.741,Z 299.095,A -85,B 0,C 180,E1 -23989.595,E2 -23989.595} C_VEL
LIN {X 0,Y 157.294,Z 286.473,A -85,B 0,C 180,E1 -23991.636,E2 -23991.636} C_VEL
LIN {X 0,Y 158.636,Z 273.07,A -85,B 0,C 180,E1 -23993.215,E2 -23993.215} C_VEL
LIN {X 0,Y 159.703,Z 258.673,A -85,B 0,C 180,E1 -23994.364,E2 -23994.364} C_VEL
LIN {X 0,Y 163.023,Z 205.225,A -85,B 0,C 180,E1 -23997.653,E2 -23997.653} C_VEL
LIN {X 0,Y 152.771,Z 176.562,A -85,B 0,C 180,E1 -24000.843,E2 -24000.843} C_VEL
LIN {X 0,Y 150.276,Z 169.771,A -85,B 0,C 180,E1 -24001.736,E2 -24001.736} C_VEL
LIN {X 0,Y 150.262,Z 169.768,A -85,B 0,C 180,E1 -24008.026,E2 -24008.026} C_VEL
LIN {X 0,Y 150.318,Z 169.76,A -85,B 0,C 180,E1 -24010.895,E2 -24010.895} C_VEL
LIN {X 0,Y 150.429,Z 169.741,A -85,B 0,C 180,E1 -24016.49,E2 -24016.49} C_VEL
LIN {X 0,Y 150.647,Z 169.72,A -85,B 0,C 180,E1 -24019.244,E2 -24019.244} C_VEL
LIN {X 0,Y 150.741,Z 169.706,A -85,B 0,C 180,E1 -24021.959,E2 -24021.959} C_VEL
LIN {X 0,Y 151.217,Z 169.648,A -85,B 0,C 180,E1 -24029.999,E2 -24029.999} C_VEL
LIN {X 0,Y 150.743,Z 169.707,A -85,B 0,C 180,E1 -24038.039,E2 -24038.039} C_VEL
LIN {X 0,Y 150.612,Z 169.718,A -85,B 0,C 180,E1 -24041.506,E2 -24041.506} C_VEL
LIN {X 0,Y 150.366,Z 169.756,A -85,B 0,C 180,E1 -24046.285,E2 -24046.285} C_VEL
LIN {X 0,Y 150.347,Z 169.755,A -85,B 0,C 180,E1 -24050.79,E2 -24050.79} C_VEL
LIN {X 0,Y 150.238,Z 169.765,A -85,B 0,C 180,E1 -24057.279,E2 -24057.279} C_VEL
LIN {X 0,Y 150.215,Z 169.773,A -85,B 0,C 180,E1 -24062.634,E2 -24062.634} C_VEL
LIN {X 0,Y 150.23,Z 169.768,A -85,B 0,C 180,E1 -24067.455,E2 -24067.455} C_VEL
LIN {X 0,Y 150.226,Z 169.772,A -85,B 0,C 180,E1 -24071.539,E2 -24071.539} C_VEL
LIN {X 0,Y 150.25,Z 169.764,A -85,B 0,C 180,E1 -24075.443,E2 -24075.443} C_VEL
LIN {X 0,Y 150.226,Z 169.771,A -85,B 0,C 180,E1 -24079.085,E2 -24079.085} C_VEL
LIN {X 0,Y 150.232,Z 169.764,A -85,B 0,C 180,E1 -24082.679,E2 -24082.679} C_VEL
LIN {X 0,Y 150.22,Z 169.774,A -85,B 0,C 180,E1 -24087.363,E2 -24087.363} C_VEL
LIN {X 0,Y 150.242,Z 169.767,A -85,B 0,C 180,E1 -24092.718,E2 -24092.718} C_VEL
LIN {X 0,Y 150.348,Z 169.752,A -85,B 0,C 180,E1 -24099.208,E2 -24099.208} C_VEL
LIN {X 0,Y 150.381,Z 169.752,A -85,B 0,C 180,E1 -24103.716,E2 -24103.716} C_VEL
LIN {X 0,Y 150.656,Z 169.717,A -85,B 0,C 180,E1 -24109.247,E2 -24109.247} C_VEL
LIN {X 0,Y 150.743,Z 169.707,A -85,B 0,C 180,E1 -24111.961,E2 -24111.961} C_VEL
LIN {X 0,Y 151.217,Z 169.648,A -85,B 0,C 180,E1 -24120.001,E2 -24120.001} C_VEL
LIN {X 0,Y 150.762,Z 169.705,A -85,B 0,C 180,E1 -24128.04,E2 -24128.04} C_VEL
LIN {X 0,Y 150.633,Z 169.716,A -85,B 0,C 180,E1 -24131.546,E2 -24131.546} C_VEL
LIN {X 0,Y 150.367,Z 169.755,A -85,B 0,C 180,E1 -24136.287,E2 -24136.287} C_VEL
LIN {X 0,Y 150.348,Z 169.752,A -85,B 0,C 180,E1 -24140.792,E2 -24140.792} C_VEL
LIN {X 0,Y 150.24,Z 169.767,A -85,B 0,C 180,E1 -24147.281,E2 -24147.281} C_VEL
LIN {X 0,Y 150.218,Z 169.773,A -85,B 0,C 180,E1 -24152.636,E2 -24152.636} C_VEL
LIN {X 0,Y 150.212,Z 169.768,A -85,B 0,C 180,E1 -24157.463,E2 -24157.463} C_VEL
LIN {X 0,Y 150.157,Z 169.781,A -85,B 0,C 180,E1 -24161.509,E2 -24161.509} C_VEL
LIN {X 0,Y 150.154,Z 169.776,A -85,B 0,C 180,E1 -24165.407,E2 -24165.407} C_VEL
LIN {X 0,Y 150.29,Z 169.827,A -85,B 0,C 180,E1 -24170.154,E2 -24170.154} C_VEL
LIN {X 0,Y 151.176,Z 174.047,A -85,B 0,C 180,E1 -24172.514,E2 -24172.514} C_VEL
LIN {X 0,Y 159.134,Z 201.317,A -85,B 0,C 180,E1 -24175.422,E2 -24175.422} C_VEL
LIN {X 0,Y 161.833,Z 237.36,A -85,B 0,C 180,E1 -24178.143,E2 -24178.143} C_VEL
LIN {X 0,Y 158.987,Z 284.417,A -85,B 0,C 180,E1 -24181.178,E2 -24181.178} C_VEL
LIN {X 0,Y 157.632,Z 298.625,A -85,B 0,C 180,E1 -24182.628,E2 -24182.628} C_VEL
LIN {X 0,Y 155.908,Z 311.682,A -85,B 0,C 180,E1 -24184.533,E2 -24184.533} C_VEL
LIN {X 0,Y 154.127,Z 323.674,A -85,B 0,C 180,E1 -24186.842,E2 -24186.842} C_VEL
LIN {X 0,Y 152.261,Z 335.293,A -85,B 0,C 180,E1 -24189.747,E2 -24189.747} C_VEL
LIN {X 0,Y 150.683,Z 345.761,A -85,B 0,C 180,E1 -24193.053,E2 -24193.053} C_VEL
LIN {X 0,Y 149.679,Z 354.302,A -85,B 0,C 180,E1 -24196.423,E2 -24196.423} C_VEL
LIN {X 0,Y 148.907,Z 362.536,A -85,B 0,C 180,E1 -24200.493,E2 -24200.493} C_VEL
LIN {X 0,Y 148.752,Z 369.116,A -85,B 0,C 180,E1 -24204.579,E2 -24204.579} C_VEL
LIN {X 0,Y 148.773,Z 374.21,A -85,B 0,C 180,E1 -24208.648,E2 -24208.648} C_VEL
LIN {X 0,Y 148.63,Z 376.834,A -85,B 0,C 180,E1 -24211.356,E2 -24211.356} C_VEL
LIN {X 0,Y 148.349,Z 378.59,A -85,B 0,C 180,E1 -24213.644,E2 -24213.644} C_VEL
LIN {X 0,Y 147.52,Z 379.935,A -85,B 0,C 180,E1 -24215.851,E2 -24215.851} C_VEL
LIN {X 0,Y 144.814,Z 381.321,A -85,B 0,C 180,E1 -24219.551,E2 -24219.551} C_VEL
LIN {X 0,Y 142.929,Z 381.997,A -85,B 0,C 180,E1 -24222.629,E2 -24222.629} C_VEL
LIN {X 0,Y 142.554,Z 382.416,A -85,B 0,C 180,E1 -24225.005,E2 -24225.005} C_VEL
LIN {X 0,Y 142.741,Z 382.512,A -85,B 0,C 180,E1 -24225.796,E2 -24225.796} C_VEL
LIN {X 0,Y 144.804,Z 382.838,A -85,B 0,C 180,E1 -24229.862,E2 -24229.862} C_VEL
LIN {X 0,Y 148.902,Z 382.03,A -85,B 0,C 180,E1 -24235.138,E2 -24235.138} C_VEL
LIN {X 0,Y 154.3,Z 379.834,A -85,B 0,C 180,E1 -24240.069,E2 -24240.069} C_VEL
LIN {X 0,Y 159.253,Z 377.218,A -85,B 0,C 180,E1 -24243.48,E2 -24243.48} C_VEL
LIN {X 0,Y 164.928,Z 373.72,A -85,B 0,C 180,E1 -24246.626,E2 -24246.626} C_VEL
LIN {X 0,Y 173.31,Z 367.653,A -85,B 0,C 180,E1 -24250.454,E2 -24250.454} C_VEL
LIN {X 0,Y 181.518,Z 360.72,A -85,B 0,C 180,E1 -24253.413,E2 -24253.413} C_VEL
LIN {X 0,Y 190.34,Z 352.052,A -85,B 0,C 180,E1 -24256.056,E2 -24256.056} C_VEL
LIN {X 0,Y 198.267,Z 342.96,A -85,B 0,C 180,E1 -24258.108,E2 -24258.108} C_VEL
LIN {X 0,Y 205.185,Z 333.778,A -85,B 0,C 180,E1 -24259.651,E2 -24259.651} C_VEL
LIN {X 0,Y 212.721,Z 322.087,A -85,B 0,C 180,E1 -24261.074,E2 -24261.074} C_VEL
LIN {X 0,Y 219.074,Z 310.234,A -85,B 0,C 180,E1 -24262.155,E2 -24262.155} C_VEL
LIN {X 0,Y 224.504,Z 297.779,A -85,B 0,C 180,E1 -24262.985,E2 -24262.985} C_VEL
LIN {X 0,Y 228.92,Z 284.66,A -85,B 0,C 180,E1 -24263.622,E2 -24263.622} C_VEL
LIN {X 0,Y 231.534,Z 274.282,A -85,B 0,C 180,E1 -24264.039,E2 -24264.039} C_VEL
LIN {X 0,Y 231.367,Z 271.551,A -85,B 0,C 180,E1 -24266.327,E2 -24266.327} C_VEL
LIN {X 0,Y 231.448,Z 270.249,A -85,B 0,C 180,E1 -24267.646,E2 -24267.646} C_VEL
LIN {X 0,Y 231.8,Z 270.356,A -85,B 0,C 180,E1 -24270.682,E2 -24270.682} C_VEL
LIN {X 0,Y 232.035,Z 270.877,A -85,B 0,C 180,E1 -24271.694,E2 -24271.694} C_VEL
LIN {X 0,Y 228.866,Z 283.535,A -85,B 0,C 180,E1 -24272.322,E2 -24272.322} C_VEL
LIN {X 0,Y 224.74,Z 295.502,A -85,B 0,C 180,E1 -24273.118,E2 -24273.118} C_VEL
LIN {X 0,Y 219.482,Z 307.473,A -85,B 0,C 180,E1 -24274.176,E2 -24274.176} C_VEL
LIN {X 0,Y 213.515,Z 318.435,A -85,B 0,C 180,E1 -24275.445,E2 -24275.445} C_VEL
LIN {X 0,Y 206.362,Z 329.386,A -85,B 0,C 180,E1 -24277.084,E2 -24277.084} C_VEL
LIN {X 0,Y 199.549,Z 338.189,A -85,B 0,C 180,E1 -24278.838,E2 -24278.838} C_VEL
LIN {X 0,Y 192.582,Z 345.863,A -85,B 0,C 180,E1 -24280.825,E2 -24280.825} C_VEL
LIN {X 0,Y 184.905,Z 353.126,A -85,B 0,C 180,E1 -24283.301,E2 -24283.301} C_VEL
LIN {X 0,Y 177.158,Z 359.324,A -85,B 0,C 180,E1 -24286.229,E2 -24286.229} C_VEL
LIN {X 0,Y 170.203,Z 363.935,A -85,B 0,C 180,E1 -24289.289,E2 -24289.289} C_VEL
LIN {X 0,Y 162.764,Z 367.929,A -85,B 0,C 180,E1 -24293.281,E2 -24293.281} C_VEL
LIN {X 0,Y 156.526,Z 370.272,A -85,B 0,C 180,E1 -24297.426,E2 -24297.426} C_VEL
LIN {X 0,Y 153.373,Z 371.036,A -85,B 0,C 180,E1 -24299.999,E2 -24299.999} C_VEL
LIN {X 0,Y 150.526,Z 371.398,A -85,B 0,C 180,E1 -24302.675,E2 -24302.675} C_VEL
LIN {X 0,Y 148.034,Z 371.281,A -85,B 0,C 180,E1 -24305.447,E2 -24305.447} C_VEL
LIN {X 0,Y 145.884,Z 370.74,A -85,B 0,C 180,E1 -24308.309,E2 -24308.309} C_VEL
LIN {X 0,Y 143.718,Z 369.452,A -85,B 0,C 180,E1 -24312.029,E2 -24312.029} C_VEL
LIN {X 0,Y 141.667,Z 366.445,A -85,B 0,C 180,E1 -24317.316,E2 -24317.316} C_VEL
LIN {X 0,Y 140.745,Z 362.646,A -85,B 0,C 180,E1 -24321.993,E2 -24321.993} C_VEL
LIN {X 0,Y 140.642,Z 357.598,A -85,B 0,C 180,E1 -24326.726,E2 -24326.726} C_VEL
LIN {X 0,Y 141.1,Z 351.661,A -85,B 0,C 180,E1 -24331.097,E2 -24331.097} C_VEL
LIN {X 0,Y 141.748,Z 345.457,A -85,B 0,C 180,E1 -24334.762,E2 -24334.762} C_VEL
LIN {X 0,Y 142.817,Z 337.376,A -85,B 0,C 180,E1 -24338.684,E2 -24338.684} C_VEL
LIN {X 0,Y 144.316,Z 327.554,A -85,B 0,C 180,E1 -24342.507,E2 -24342.507} C_VEL
LIN {X 0,Y 145.956,Z 317.202,A -85,B 0,C 180,E1 -24345.752,E2 -24345.752} C_VEL
LIN {X 0,Y 147.659,Z 305.991,A -85,B 0,C 180,E1 -24348.552,E2 -24348.552} C_VEL
LIN {X 0,Y 149.574,Z 292.864,A -85,B 0,C 180,E1 -24351.096,E2 -24351.096} C_VEL
LIN {X 0,Y 151.051,Z 280.352,A -85,B 0,C 180,E1 -24352.917,E2 -24352.917} C_VEL
LIN {X 0,Y 152.274,Z 265.78,A -85,B 0,C 180,E1 -24354.432,E2 -24354.432} C_VEL
LIN {X 0,Y 156.097,Z 206.388,A -85,B 0,C 180,E1 -24358.32,E2 -24358.32} C_VEL
LIN {X 0,Y 146.201,Z 178.784,A -85,B 0,C 180,E1 -24361.524,E2 -24361.524} C_VEL
LIN {X 0,Y 143.261,Z 170.644,A -85,B 0,C 180,E1 -24362.579,E2 -24362.579} C_VEL
LIN {X 0,Y 143.284,Z 170.635,A -85,B 0,C 180,E1 -24369.918,E2 -24369.918} C_VEL
LIN {X 0,Y 143.348,Z 170.623,A -85,B 0,C 180,E1 -24375.809,E2 -24375.809} C_VEL
LIN {X 0,Y 143.593,Z 170.596,A -85,B 0,C 180,E1 -24378.709,E2 -24378.709} C_VEL
LIN {X 0,Y 143.66,Z 170.589,A -85,B 0,C 180,E1 -24381.56,E2 -24381.56} C_VEL
LIN {X 0,Y 144.176,Z 170.525,A -85,B 0,C 180,E1 -24389.999,E2 -24389.999} C_VEL
LIN {X 0,Y 143.663,Z 170.59,A -85,B 0,C 180,E1 -24398.438,E2 -24398.438} C_VEL
LIN {X 0,Y 143.546,Z 170.598,A -85,B 0,C 180,E1 -24401.712,E2 -24401.712} C_VEL
LIN {X 0,Y 143.303,Z 170.633,A -85,B 0,C 180,E1 -24407.112,E2 -24407.112} C_VEL
LIN {X 0,Y 143.273,Z 170.635,A -85,B 0,C 180,E1 -24411.252,E2 -24411.252} C_VEL
LIN {X 0,Y 143.185,Z 170.644,A -85,B 0,C 180,E1 -24417.935,E2 -24417.935} C_VEL
LIN {X 0,Y 143.166,Z 170.651,A -85,B 0,C 180,E1 -24423.435,E2 -24423.435} C_VEL
LIN {X 0,Y 143.121,Z 170.657,A -85,B 0,C 180,E1 -24429.669,E2 -24429.669} C_VEL
LIN {X 0,Y 143.159,Z 170.65,A -85,B 0,C 180,E1 -24433.415,E2 -24433.415} C_VEL
LIN {X 0,Y 143.154,Z 170.652,A -85,B 0,C 180,E1 -24437.425,E2 -24437.425} C_VEL
LIN {X 0,Y 143.136,Z 170.65,A -85,B 0,C 180,E1 -24441.775,E2 -24441.775} C_VEL
LIN {X 0,Y 143.187,Z 170.65,A -85,B 0,C 180,E1 -24447.324,E2 -24447.324} C_VEL
LIN {X 0,Y 143.189,Z 170.646,A -85,B 0,C 180,E1 -24452.062,E2 -24452.062} C_VEL
LIN {X 0,Y 143.274,Z 170.634,A -85,B 0,C 180,E1 -24458.746,E2 -24458.746} C_VEL
LIN {X 0,Y 143.314,Z 170.633,A -85,B 0,C 180,E1 -24462.889,E2 -24462.889} C_VEL
LIN {X 0,Y 143.592,Z 170.594,A -85,B 0,C 180,E1 -24468.711,E2 -24468.711} C_VEL
LIN {X 0,Y 143.663,Z 170.589,A -85,B 0,C 180,E1 -24471.562,E2 -24471.562} C_VEL
LIN {X 0,Y 144.176,Z 170.525,A -85,B 0,C 180,E1 -24480.001,E2 -24480.001} C_VEL
LIN {X 0,Y 143.684,Z 170.588,A -85,B 0,C 180,E1 -24488.439,E2 -24488.439} C_VEL
LIN {X 0,Y 143.57,Z 170.596,A -85,B 0,C 180,E1 -24491.759,E2 -24491.759} C_VEL
LIN {X 0,Y 143.304,Z 170.634,A -85,B 0,C 180,E1 -24497.114,E2 -24497.114} C_VEL
LIN {X 0,Y 143.274,Z 170.633,A -85,B 0,C 180,E1 -24501.254,E2 -24501.254} C_VEL
LIN {X 0,Y 143.188,Z 170.646,A -85,B 0,C 180,E1 -24507.937,E2 -24507.937} C_VEL
LIN {X 0,Y 143.169,Z 170.651,A -85,B 0,C 180,E1 -24513.437,E2 -24513.437} C_VEL
LIN {X 0,Y 143.078,Z 170.661,A -85,B 0,C 180,E1 -24519.686,E2 -24519.686} C_VEL
LIN {X 0,Y 143.073,Z 170.662,A -85,B 0,C 180,E1 -24523.45,E2 -24523.45} C_VEL
LIN {X 0,Y 143.234,Z 170.75,A -85,B 0,C 180,E1 -24529.794,E2 -24529.794} C_VEL
LIN {X 0,Y 143.878,Z 173.589,A -85,B 0,C 180,E1 -24531.475,E2 -24531.475} C_VEL
LIN {X 0,Y 152.394,Z 202.606,A -85,B 0,C 180,E1 -24534.748,E2 -24534.748} C_VEL
LIN {X 0,Y 154.96,Z 237.37,A -85,B 0,C 180,E1 -24537.511,E2 -24537.511} C_VEL
LIN {X 0,Y 152.021,Z 284.248,A -85,B 0,C 180,E1 -24540.677,E2 -24540.677} C_VEL
LIN {X 0,Y 150.651,Z 298.386,A -85,B 0,C 180,E1 -24542.193,E2 -24542.193} C_VEL
LIN {X 0,Y 148.772,Z 312.14,A -85,B 0,C 180,E1 -24544.314,E2 -24544.314} C_VEL
LIN {X 0,Y 146.959,Z 324.034,A -85,B 0,C 180,E1 -24546.764,E2 -24546.764} C_VEL
LIN {X 0,Y 145.072,Z 335.43,A -85,B 0,C 180,E1 -24549.809,E2 -24549.809} C_VEL
LIN {X 0,Y 143.662,Z 344.787,A -85,B 0,C 180,E1 -24552.932,E2 -24552.932} C_VEL
LIN {X 0,Y 142.645,Z 353.406,A -85,B 0,C 180,E1 -24556.467,E2 -24556.467} C_VEL
LIN {X 0,Y 141.896,Z 361.709,A -85,B 0,C 180,E1 -24560.738,E2 -24560.738} C_VEL
LIN {X 0,Y 141.764,Z 367.354,A -85,B 0,C 180,E1 -24564.311,E2 -24564.311} C_VEL
LIN {X 0,Y 141.78,Z 372.722,A -85,B 0,C 180,E1 -24568.581,E2 -24568.581} C_VEL
LIN {X 0,Y 141.68,Z 375.538,A -85,B 0,C 180,E1 -24571.422,E2 -24571.422} C_VEL
LIN {X 0,Y 141.215,Z 378.674,A -85,B 0,C 180,E1 -24575.714,E2 -24575.714} C_VEL
LIN {X 0,Y 141.271,Z 380.26,A -85,B 0,C 180,E1 -24578.584,E2 -24578.584} C_VEL
LIN {X 0,Y 142.258,Z 382.275,A -85,B 0,C 180,E1 -24584.302,E2 -24584.302} C_VEL
LIN {X 0,Y 142.741,Z 382.512,A -85,B 0,C 180,E1 -24585.796,E2 -24585.796} C_VEL
LIN {X 0,Y 143.094,Z 382.753,A -85,B 0,C 180,E1 -24588.16,E2 -24588.16} C_VEL
LIN {X 0,Y 142.621,Z 382.547,A -85,B 0,C 180,E1 -24592.132,E2 -24592.132} C_VEL
LIN {X 0,Y 142.706,Z 382.049,A -85,B 0,C 180,E1 -24595.309,E2 -24595.309} C_VEL
LIN {X 0,Y 143.841,Z 381.486,A -85,B 0,C 180,E1 -24597.615,E2 -24597.615} C_VEL
LIN {X 0,Y 144.521,Z 381.225,A -85,B 0,C 180,E1 -24598.344,E2 -24598.344} C_VEL
LIN {X 0,Y 148.191,Z 379.92,A -85,B 0,C 180,E1 -24601.446,E2 -24601.446} C_VEL
LIN {X 0,Y 155.288,Z 376.609,A -85,B 0,C 180,E1 -24606.041,E2 -24606.041} C_VEL
LIN {X 0,Y 161.396,Z 373.136,A -85,B 0,C 180,E1 -24609.155,E2 -24609.155} C_VEL
LIN {X 0,Y 168.044,Z 368.73,A -85,B 0,C 180,E1 -24612.003,E2 -24612.003} C_VEL
LIN {X 0,Y 176.53,Z 362.263,A -85,B 0,C 180,E1 -24614.965,E2 -24614.965} C_VEL
LIN {X 0,Y 185.624,Z 354.183,A -85,B 0,C 180,E1 -24617.588,E2 -24617.588} C_VEL
LIN {X 0,Y 193.776,Z 345.631,A -85,B 0,C 180,E1 -24619.61,E2 -24619.61} C_VEL
LIN {X 0,Y 202.279,Z 335.29,A -85,B 0,C 180,E1 -24621.422,E2 -24621.422} C_VEL
LIN {X 0,Y 209.565,Z 324.849,A -85,B 0,C 180,E1 -24622.717,E2 -24622.717} C_VEL
LIN {X 0,Y 216.761,Z 312.444,A -85,B 0,C 180,E1 -24623.857,E2 -24623.857} C_VEL
LIN {X 0,Y 222.356,Z 300.524,A -85,B 0,C 180,E1 -24624.638,E2 -24624.638} C_VEL
LIN {X 0,Y 227.144,Z 287.698,A -85,B 0,C 180,E1 -24625.281,E2 -24625.281} C_VEL
LIN {X 0,Y 229.614,Z 279.347,A -85,B 0,C 180,E1 -24625.65,E2 -24625.65} C_VEL
LIN {X 0,Y 229.779,Z 277.128,A -85,B 0,C 180,E1 -24627.952,E2 -24627.952} C_VEL
LIN {X 0,Y 230.008,Z 277.264,A -85,B 0,C 180,E1 -24630.223,E2 -24630.223} C_VEL
LIN {X 0,Y 226.378,Z 289.178,A -85,B 0,C 180,E1 -24630.838,E2 -24630.838} C_VEL
LIN {X 0,Y 221.15,Z 302.089,A -85,B 0,C 180,E1 -24631.788,E2 -24631.788} C_VEL
LIN {X 0,Y 215.596,Z 313.171,A -85,B 0,C 180,E1 -24632.846,E2 -24632.846} C_VEL
LIN {X 0,Y 209.33,Z 323.429,A -85,B 0,C 180,E1 -24634.121,E2 -24634.121} C_VEL
LIN {X 0,Y 202.061,Z 333.293,A -85,B 0,C 180,E1 -24635.69,E2 -24635.69} C_VEL
LIN {X 0,Y 194.142,Z 342.471,A -85,B 0,C 180,E1 -24637.659,E2 -24637.659} C_VEL
LIN {X 0,Y 187.643,Z 348.9,A -85,B 0,C 180,E1 -24639.449,E2 -24639.449} C_VEL
LIN {X 0,Y 180.09,Z 355.345,A -85,B 0,C 180,E1 -24641.807,E2 -24641.807} C_VEL
LIN {X 0,Y 172.316,Z 360.978,A -85,B 0,C 180,E1 -24644.626,E2 -24644.626} C_VEL
LIN {X 0,Y 165.026,Z 365.329,A -85,B 0,C 180,E1 -24647.705,E2 -24647.705} C_VEL
LIN {X 0,Y 160.532,Z 367.546,A -85,B 0,C 180,E1 -24649.914,E2 -24649.914} C_VEL
LIN {X 0,Y 155.963,Z 369.457,A -85,B 0,C 180,E1 -24652.471,E2 -24652.471} C_VEL
LIN {X 0,Y 152.44,Z 370.607,A -85,B 0,C 180,E1 -24654.708,E2 -24654.708} C_VEL
LIN {X 0,Y 147.657,Z 371.661,A -85,B 0,C 180,E1 -24658.277,E2 -24658.277} C_VEL
LIN {X 0,Y 142.861,Z 371.845,A -85,B 0,C 180,E1 -24662.819,E2 -24662.819} C_VEL
LIN {X 0,Y 140.36,Z 371.375,A -85,B 0,C 180,E1 -24665.746,E2 -24665.746} C_VEL
LIN {X 0,Y 138.257,Z 370.481,A -85,B 0,C 180,E1 -24668.771,E2 -24668.771} C_VEL
LIN {X 0,Y 136.514,Z 369.117,A -85,B 0,C 180,E1 -24671.993,E2 -24671.993} C_VEL
LIN {X 0,Y 134.712,Z 366.319,A -85,B 0,C 180,E1 -24676.674,E2 -24676.674} C_VEL
LIN {X 0,Y 133.705,Z 362.333,A -85,B 0,C 180,E1 -24681.588,E2 -24681.588} C_VEL
LIN {X 0,Y 133.628,Z 356.198,A -85,B 0,C 180,E1 -24687.245,E2 -24687.245} C_VEL
LIN {X 0,Y 134.12,Z 350.179,A -85,B 0,C 180,E1 -24691.6,E2 -24691.6} C_VEL
LIN {X 0,Y 134.938,Z 342.894,A -85,B 0,C 180,E1 -24695.868,E2 -24695.868} C_VEL
LIN {X 0,Y 135.981,Z 335.276,A -85,B 0,C 180,E1 -24699.523,E2 -24699.523} C_VEL
LIN {X 0,Y 137.452,Z 326.023,A -85,B 0,C 180,E1 -24703.145,E2 -24703.145} C_VEL
LIN {X 0,Y 139.155,Z 315.142,A -85,B 0,C 180,E1 -24706.551,E2 -24706.551} C_VEL
LIN {X 0,Y 141.184,Z 302.452,A -85,B 0,C 180,E1 -24709.673,E2 -24709.673} C_VEL
LIN {X 0,Y 142.974,Z 289.161,A -85,B 0,C 180,E1 -24712.143,E2 -24712.143} C_VEL
LIN {X 0,Y 144.513,Z 275.911,A -85,B 0,C 180,E1 -24713.961,E2 -24713.961} C_VEL
LIN {X 0,Y 145.615,Z 261.872,A -85,B 0,C 180,E1 -24715.283,E2 -24715.283} C_VEL
LIN {X 0,Y 149.22,Z 207.653,A -85,B 0,C 180,E1 -24718.985,E2 -24718.985} C_VEL
LIN {X 0,Y 138.904,Z 178.979,A -85,B 0,C 180,E1 -24722.522,E2 -24722.522} C_VEL
LIN {X 0,Y 136.168,Z 171.526,A -85,B 0,C 180,E1 -24723.565,E2 -24723.565} C_VEL
LIN {X 0,Y 136.234,Z 171.516,A -85,B 0,C 180,E1 -24728.83,E2 -24728.83} C_VEL
LIN {X 0,Y 136.253,Z 171.509,A -85,B 0,C 180,E1 -24735.053,E2 -24735.053} C_VEL
LIN {X 0,Y 136.496,Z 171.479,A -85,B 0,C 180,E1 -24738.114,E2 -24738.114} C_VEL
LIN {X 0,Y 136.588,Z 171.471,A -85,B 0,C 180,E1 -24741.119,E2 -24741.119} C_VEL
LIN {X 0,Y 137.133,Z 171.402,A -85,B 0,C 180,E1 -24749.999,E2 -24749.999} C_VEL
LIN {X 0,Y 136.59,Z 171.469,A -85,B 0,C 180,E1 -24758.879,E2 -24758.879} C_VEL
LIN {X 0,Y 136.489,Z 171.477,A -85,B 0,C 180,E1 -24761.953,E2 -24761.953} C_VEL
LIN {X 0,Y 136.241,Z 171.512,A -85,B 0,C 180,E1 -24768.028,E2 -24768.028} C_VEL
LIN {X 0,Y 136.194,Z 171.518,A -85,B 0,C 180,E1 -24771.746,E2 -24771.746} C_VEL
LIN {X 0,Y 136.096,Z 171.528,A -85,B 0,C 180,E1 -24778.615,E2 -24778.615} C_VEL
LIN {X 0,Y 136.079,Z 171.531,A -85,B 0,C 180,E1 -24784.617,E2 -24784.617} C_VEL
LIN {X 0,Y 136.087,Z 171.532,A -85,B 0,C 180,E1 -24789.228,E2 -24789.228} C_VEL
LIN {X 0,Y 136.094,Z 171.528,A -85,B 0,C 180,E1 -24793.701,E2 -24793.701} C_VEL
LIN {X 0,Y 136.103,Z 171.532,A -85,B 0,C 180,E1 -24797.835,E2 -24797.835} C_VEL
LIN {X 0,Y 136.088,Z 171.528,A -85,B 0,C 180,E1 -24801.706,E2 -24801.706} C_VEL
LIN {X 0,Y 136.091,Z 171.533,A -85,B 0,C 180,E1 -24805.716,E2 -24805.716} C_VEL
LIN {X 0,Y 136.145,Z 171.523,A -85,B 0,C 180,E1 -24812.317,E2 -24812.317} C_VEL
LIN {X 0,Y 136.241,Z 171.509,A -85,B 0,C 180,E1 -24818.834,E2 -24818.834} C_VEL
LIN {X 0,Y 136.281,Z 171.509,A -85,B 0,C 180,E1 -24825.059,E2 -24825.059} C_VEL
LIN {X 0,Y 136.495,Z 171.477,A -85,B 0,C 180,E1 -24828.116,E2 -24828.116} C_VEL
LIN {X 0,Y 136.59,Z 171.472,A -85,B 0,C 180,E1 -24831.121,E2 -24831.121} C_VEL
LIN {X 0,Y 137.133,Z 171.402,A -85,B 0,C 180,E1 -24840.001,E2 -24840.001} C_VEL
LIN {X 0,Y 136.607,Z 171.469,A -85,B 0,C 180,E1 -24848.88,E2 -24848.88} C_VEL
LIN {X 0,Y 136.491,Z 171.478,A -85,B 0,C 180,E1 -24851.957,E2 -24851.957} C_VEL
LIN {X 0,Y 136.243,Z 171.514,A -85,B 0,C 180,E1 -24858.031,E2 -24858.031} C_VEL
LIN {X 0,Y 136.195,Z 171.515,A -85,B 0,C 180,E1 -24861.748,E2 -24861.748} C_VEL
LIN {X 0,Y 136.098,Z 171.526,A -85,B 0,C 180,E1 -24868.617,E2 -24868.617} C_VEL
LIN {X 0,Y 136.079,Z 171.533,A -85,B 0,C 180,E1 -24874.62,E2 -24874.62} C_VEL
LIN {X 0,Y 136.053,Z 171.535,A -85,B 0,C 180,E1 -24879.211,E2 -24879.211} C_VEL
LIN {X 0,Y 136.015,Z 171.541,A -85,B 0,C 180,E1 -24883.667,E2 -24883.667} C_VEL
LIN {X 0,Y 136.152,Z 171.638,A -85,B 0,C 180,E1 -24889.416,E2 -24889.416} C_VEL
LIN {X 0,Y 136.49,Z 173.121,A -85,B 0,C 180,E1 -24890.363,E2 -24890.363} C_VEL
LIN {X 0,Y 144.559,Z 200.182,A -85,B 0,C 180,E1 -24893.633,E2 -24893.633} C_VEL
LIN {X 0,Y 145.743,Z 205.342,A -85,B 0,C 180,E1 -24894.169,E2 -24894.169} C_VEL
LIN {X 0,Y 148.05,Z 238.174,A -85,B 0,C 180,E1 -24896.885,E2 -24896.885} C_VEL
LIN {X 0,Y 145.099,Z 283.698,A -85,B 0,C 180,E1 -24900.135,E2 -24900.135} C_VEL
LIN {X 0,Y 143.731,Z 297.335,A -85,B 0,C 180,E1 -24901.662,E2 -24901.662} C_VEL
LIN {X 0,Y 142.071,Z 309.476,A -85,B 0,C 180,E1 -24903.564,E2 -24903.564} C_VEL
LIN {X 0,Y 140.029,Z 322.672,A -85,B 0,C 180,E1 -24906.328,E2 -24906.328} C_VEL
LIN {X 0,Y 138.122,Z 334.271,A -85,B 0,C 180,E1 -24909.525,E2 -24909.525} C_VEL
LIN {X 0,Y 136.639,Z 343.729,A -85,B 0,C 180,E1 -24912.799,E2 -24912.799} C_VEL
LIN {X 0,Y 135.618,Z 352.466,A -85,B 0,C 180,E1 -24916.516,E2 -24916.516} C_VEL
LIN {X 0,Y 134.88,Z 360.879,A -85,B 0,C 180,E1 -24921.008,E2 -24921.008} C_VEL
LIN {X 0,Y 134.779,Z 367.583,A -85,B 0,C 180,E1 -24925.515,E2 -24925.515} C_VEL
LIN {X 0,Y 134.85,Z 372.727,A -85,B 0,C 180,E1 -24930.001,E2 -24930.001} C_VEL
LIN {X 0,Y 134.516,Z 375.366,A -85,B 0,C 180,E1 -24932.996,E2 -24932.996} C_VEL
LIN {X 0,Y 134.245,Z 377.49,A -85,B 0,C 180,E1 -24936.011,E2 -24936.011} C_VEL
LIN {X 0,Y 134.306,Z 379.196,A -85,B 0,C 180,E1 -24939.033,E2 -24939.033} C_VEL
LIN {X 0,Y 135.395,Z 381.462,A -85,B 0,C 180,E1 -24945.044,E2 -24945.044} C_VEL
LIN {X 0,Y 138.149,Z 382.344,A -85,B 0,C 180,E1 -24950.862,E2 -24950.862} C_VEL
LIN {X 0,Y 142.5,Z 381.819,A -85,B 0,C 180,E1 -24956.352,E2 -24956.352} C_VEL
LIN {X 0,Y 144.521,Z 381.225,A -85,B 0,C 180,E1 -24958.344,E2 -24958.344} C_VEL
LIN {X 0,Y 146.335,Z 380.488,A -85,B 0,C 180,E1 -24960.538,E2 -24960.538} C_VEL
LIN {X 0,Y 148.248,Z 378.873,A -85,B 0,C 180,E1 -24964.266,E2 -24964.266} C_VEL
LIN {X 0,Y 150.84,Z 376.704,A -85,B 0,C 180,E1 -24967.816,E2 -24967.816} C_VEL
LIN {X 0,Y 153.622,Z 375.094,A -85,B 0,C 180,E1 -24969.667,E2 -24969.667} C_VEL
LIN {X 0,Y 162.904,Z 369.772,A -85,B 0,C 180,E1 -24973.653,E2 -24973.653} C_VEL
LIN {X 0,Y 170.391,Z 364.717,A -85,B 0,C 180,E1 -24976.205,E2 -24976.205} C_VEL
LIN {X 0,Y 179.655,Z 357.385,A -85,B 0,C 180,E1 -24978.856,E2 -24978.856} C_VEL
LIN {X 0,Y 189.4,Z 348.255,A -85,B 0,C 180,E1 -24981.192,E2 -24981.192} C_VEL
LIN {X 0,Y 196.6,Z 340.397,A -85,B 0,C 180,E1 -24982.694,E2 -24982.694} C_VEL
LIN {X 0,Y 204.919,Z 329.861,A -85,B 0,C 180,E1 -24984.125,E2 -24984.125} C_VEL
LIN {X 0,Y 212.653,Z 318.1,A -85,B 0,C 180,E1 -24985.296,E2 -24985.296} C_VEL
LIN {X 0,Y 219.011,Z 306.464,A -85,B 0,C 180,E1 -24986.133,E2 -24986.133} C_VEL
LIN {X 0,Y 224.228,Z 294.536,A -85,B 0,C 180,E1 -24986.789,E2 -24986.789} C_VEL
LIN {X 0,Y 227.373,Z 285.711,A -85,B 0,C 180,E1 -24987.147,E2 -24987.147} C_VEL
LIN {X 0,Y 227.678,Z 284.68,A -85,B 0,C 180,E1 -24987.333,E2 -24987.333} C_VEL
LIN {X 0,Y 227.82,Z 283.921,A -85,B 0,C 180,E1 -24988.369,E2 -24988.369} C_VEL
LIN {X 0,Y 227.844,Z 283.891,A -85,B 0,C 180,E1 -24988.582,E2 -24988.582} C_VEL
LIN {X 0,Y 227.658,Z 284.545,A -85,B 0,C 180,E1 -24988.754,E2 -24988.754} C_VEL
LIN {X 0,Y 222.929,Z 297.271,A -85,B 0,C 180,E1 -24989.53,E2 -24989.53} C_VEL
LIN {X 0,Y 217.131,Z 309.422,A -85,B 0,C 180,E1 -24990.503,E2 -24990.503} C_VEL
LIN {X 0,Y 210.863,Z 319.966,A -85,B 0,C 180,E1 -24991.643,E2 -24991.643} C_VEL
LIN {X 0,Y 202.749,Z 331.321,A -85,B 0,C 180,E1 -24993.215,E2 -24993.215} C_VEL
LIN {X 0,Y 194.925,Z 340.406,A -85,B 0,C 180,E1 -24994.926,E2 -24994.926} C_VEL
LIN {X 0,Y 187.284,Z 347.887,A -85,B 0,C 180,E1 -24996.794,E2 -24996.794} C_VEL
LIN {X 0,Y 178.553,Z 355.195,A -85,B 0,C 180,E1 -24999.252,E2 -24999.252} C_VEL
LIN {X 0,Y 169.868,Z 361.233,A -85,B 0,C 180,E1 -25002.101,E2 -25002.101} C_VEL
LIN {X 0,Y 161.2,Z 366.049,A -85,B 0,C 180,E1 -25005.498,E2 -25005.498} C_VEL
LIN {X 0,Y 153.005,Z 369.576,A -85,B 0,C 180,E1 -25009.412,E2 -25009.412} C_VEL
LIN {X 0,Y 148.744,Z 370.948,A -85,B 0,C 180,E1 -25011.85,E2 -25011.85} C_VEL
LIN {X 0,Y 144.786,Z 371.838,A -85,B 0,C 180,E1 -25014.428,E2 -25014.428} C_VEL
LIN {X 0,Y 140.689,Z 372.35,A -85,B 0,C 180,E1 -25017.568,E2 -25017.568} C_VEL
LIN {X 0,Y 135.145,Z 371.998,A -85,B 0,C 180,E1 -25022.98,E2 -25022.98} C_VEL
LIN {X 0,Y 132.685,Z 371.172,A -85,B 0,C 180,E1 -25026.08,E2 -25026.08} C_VEL
LIN {X 0,Y 129.313,Z 368.596,A -85,B 0,C 180,E1 -25031.959,E2 -25031.959} C_VEL
LIN {X 0,Y 127.308,Z 364.831,A -85,B 0,C 180,E1 -25037.674,E2 -25037.674} C_VEL
LIN {X 0,Y 126.57,Z 360.253,A -85,B 0,C 180,E1 -25042.871,E2 -25042.871} C_VEL
LIN {X 0,Y 126.677,Z 353.844,A -85,B 0,C 180,E1 -25048.459,E2 -25048.459} C_VEL
LIN {X 0,Y 127.402,Z 346.499,A -85,B 0,C 180,E1 -25053.478,E2 -25053.478} C_VEL
LIN {X 0,Y 128.437,Z 338.24,A -85,B 0,C 180,E1 -25057.994,E2 -25057.994} C_VEL
LIN {X 0,Y 130.01,Z 327.826,A -85,B 0,C 180,E1 -25062.508,E2 -25062.508} C_VEL
LIN {X 0,Y 131.806,Z 316.885,A -85,B 0,C 180,E1 -25066.274,E2 -25066.274} C_VEL
LIN {X 0,Y 133.81,Z 304.466,A -85,B 0,C 180,E1 -25069.601,E2 -25069.601} C_VEL
LIN {X 0,Y 135.723,Z 291.592,A -85,B 0,C 180,E1 -25072.223,E2 -25072.223} C_VEL
LIN {X 0,Y 137.333,Z 278.043,A -85,B 0,C 180,E1 -25074.267,E2 -25074.267} C_VEL
LIN {X 0,Y 138.536,Z 264.434,A -85,B 0,C 180,E1 -25075.69,E2 -25075.69} C_VEL
LIN {X 0,Y 142.332,Z 209.018,A -85,B 0,C 180,E1 -25079.68,E2 -25079.68} C_VEL
LIN {X 0,Y 132.64,Z 181.873,A -85,B 0,C 180,E1 -25083.229,E2 -25083.229} C_VEL
LIN {X 0,Y 129.055,Z 172.415,A -85,B 0,C 180,E1 -25084.604,E2 -25084.604} C_VEL
LIN {X 0,Y 129.105,Z 172.404,A -85,B 0,C 180,E1 -25087.728,E2 -25087.728} C_VEL
LIN {X 0,Y 129.17,Z 172.393,A -85,B 0,C 180,E1 -25094.213,E2 -25094.213} C_VEL
LIN {X 0,Y 129.415,Z 172.361,A -85,B 0,C 180,E1 -25097.819,E2 -25097.819} C_VEL
LIN {X 0,Y 129.514,Z 172.352,A -85,B 0,C 180,E1 -25100.63,E2 -25100.63} C_VEL
LIN {X 0,Y 130.088,Z 172.28,A -85,B 0,C 180,E1 -25109.999,E2 -25109.999} C_VEL
LIN {X 0,Y 129.515,Z 172.349,A -85,B 0,C 180,E1 -25119.368,E2 -25119.368} C_VEL
LIN {X 0,Y 129.391,Z 172.363,A -85,B 0,C 180,E1 -25122.547,E2 -25122.547} C_VEL
LIN {X 0,Y 129.151,Z 172.391,A -85,B 0,C 180,E1 -25129.055,E2 -25129.055} C_VEL
LIN {X 0,Y 129.105,Z 172.403,A -85,B 0,C 180,E1 -25132.398,E2 -25132.398} C_VEL
LIN {X 0,Y 129.024,Z 172.412,A -85,B 0,C 180,E1 -25135.832,E2 -25135.832} C_VEL
LIN {X 0,Y 129.013,Z 172.411,A -85,B 0,C 180,E1 -25139.357,E2 -25139.357} C_VEL
LIN {X 0,Y 129.021,Z 172.409,A -85,B 0,C 180,E1 -25145.209,E2 -25145.209} C_VEL
LIN {X 0,Y 129.012,Z 172.414,A -85,B 0,C 180,E1 -25150.82,E2 -25150.82} C_VEL
LIN {X 0,Y 129.022,Z 172.407,A -85,B 0,C 180,E1 -25155.081,E2 -25155.081} C_VEL
LIN {X 0,Y 129.011,Z 172.415,A -85,B 0,C 180,E1 -25159.698,E2 -25159.698} C_VEL
LIN {X 0,Y 129.022,Z 172.411,A -85,B 0,C 180,E1 -25164.79,E2 -25164.79} C_VEL
LIN {X 0,Y 129.048,Z 172.404,A -85,B 0,C 180,E1 -25170.651,E2 -25170.651} C_VEL
LIN {X 0,Y 129.105,Z 172.399,A -85,B 0,C 180,E1 -25177.728,E2 -25177.728} C_VEL
LIN {X 0,Y 129.157,Z 172.393,A -85,B 0,C 180,E1 -25180.946,E2 -25180.946} C_VEL
LIN {X 0,Y 129.414,Z 172.359,A -85,B 0,C 180,E1 -25187.821,E2 -25187.821} C_VEL
LIN {X 0,Y 129.515,Z 172.351,A -85,B 0,C 180,E1 -25190.632,E2 -25190.632} C_VEL
LIN {X 0,Y 130.088,Z 172.28,A -85,B 0,C 180,E1 -25200.001,E2 -25200.001} C_VEL
LIN {X 0,Y 129.529,Z 172.349,A -85,B 0,C 180,E1 -25209.369,E2 -25209.369} C_VEL
LIN {X 0,Y 129.392,Z 172.362,A -85,B 0,C 180,E1 -25212.549,E2 -25212.549} C_VEL
LIN {X 0,Y 129.153,Z 172.393,A -85,B 0,C 180,E1 -25219.058,E2 -25219.058} C_VEL
LIN {X 0,Y 129.107,Z 172.4,A -85,B 0,C 180,E1 -25222.4,E2 -25222.4} C_VEL
LIN {X 0,Y 129.027,Z 172.413,A -85,B 0,C 180,E1 -25225.835,E2 -25225.835} C_VEL
LIN {X 0,Y 129.016,Z 172.408,A -85,B 0,C 180,E1 -25229.359,E2 -25229.359} C_VEL
LIN {X 0,Y 128.992,Z 172.415,A -85,B 0,C 180,E1 -25235.191,E2 -25235.191} C_VEL
LIN {X 0,Y 128.977,Z 172.418,A -85,B 0,C 180,E1 -25240.837,E2 -25240.837} C_VEL
LIN {X 0,Y 129.012,Z 172.415,A -85,B 0,C 180,E1 -25247.344,E2 -25247.344} C_VEL
LIN {X 0,Y 129.092,Z 172.514,A -85,B 0,C 180,E1 -25249.024,E2 -25249.024} C_VEL
LIN {X 0,Y 133.391,Z 186.345,A -85,B 0,C 180,E1 -25251,E2 -25251} C_VEL
LIN {X 0,Y 138.939,Z 205.854,A -85,B 0,C 180,E1 -25253.383,E2 -25253.383} C_VEL
LIN {X 0,Y 141.144,Z 238.65,A -85,B 0,C 180,E1 -25256.241,E2 -25256.241} C_VEL
LIN {X 0,Y 138.141,Z 283.451,A -85,B 0,C 180,E1 -25259.606,E2 -25259.606} C_VEL
LIN {X 0,Y 136.691,Z 297.486,A -85,B 0,C 180,E1 -25261.269,E2 -25261.269} C_VEL
LIN {X 0,Y 134.96,Z 309.706,A -85,B 0,C 180,E1 -25263.312,E2 -25263.312} C_VEL
LIN {X 0,Y 133.124,Z 321.272,A -85,B 0,C 180,E1 -25265.85,E2 -25265.85} C_VEL
LIN {X 0,Y 131.144,Z 333.095,A -85,B 0,C 180,E1 -25269.206,E2 -25269.206} C_VEL
LIN {X 0,Y 129.643,Z 342.682,A -85,B 0,C 180,E1 -25272.654,E2 -25272.654} C_VEL
LIN {X 0,Y 128.604,Z 351.475,A -85,B 0,C 180,E1 -25276.571,E2 -25276.571} C_VEL
LIN {X 0,Y 127.937,Z 358.666,A -85,B 0,C 180,E1 -25280.516,E2 -25280.516} C_VEL
LIN {X 0,Y 127.802,Z 365.707,A -85,B 0,C 180,E1 -25285.27,E2 -25285.27} C_VEL
LIN {X 0,Y 127.879,Z 371.151,A -85,B 0,C 180,E1 -25290.001,E2 -25290.001} C_VEL
LIN {X 0,Y 127.566,Z 373.929,A -85,B 0,C 180,E1 -25293.159,E2 -25293.159} C_VEL
LIN {X 0,Y 127.285,Z 376.212,A -85,B 0,C 180,E1 -25296.341,E2 -25296.341} C_VEL
LIN {X 0,Y 127.743,Z 379.518,A -85,B 0,C 180,E1 -25302.714,E2 -25302.714} C_VEL
LIN {X 0,Y 129.753,Z 381.332,A -85,B 0,C 180,E1 -25308.966,E2 -25308.966} C_VEL
LIN {X 0,Y 133.64,Z 381.802,A -85,B 0,C 180,E1 -25314.881,E2 -25314.881} C_VEL
LIN {X 0,Y 138.999,Z 380.926,A -85,B 0,C 180,E1 -25320.373,E2 -25320.373} C_VEL
LIN {X 0,Y 145.719,Z 378.687,A -85,B 0,C 180,E1 -25325.364,E2 -25325.364} C_VEL
LIN {X 0,Y 153.622,Z 375.094,A -85,B 0,C 180,E1 -25329.667,E2 -25329.667} C_VEL
LIN {X 0,Y 155.427,Z 373.984,A -85,B 0,C 180,E1 -25330.928,E2 -25330.928} C_VEL
LIN {X 0,Y 158.987,Z 370.341,A -85,B 0,C 180,E1 -25335.493,E2 -25335.493} C_VEL
LIN {X 0,Y 161.129,Z 368.847,A -85,B 0,C 180,E1 -25336.561,E2 -25336.561} C_VEL
LIN {X 0,Y 170.996,Z 362.338,A -85,B 0,C 180,E1 -25339.497,E2 -25339.497} C_VEL
LIN {X 0,Y 180.843,Z 354.62,A -85,B 0,C 180,E1 -25341.904,E2 -25341.904} C_VEL
LIN {X 0,Y 189.544,Z 346.516,A -85,B 0,C 180,E1 -25343.752,E2 -25343.752} C_VEL
LIN {X 0,Y 198.705,Z 336.515,A -85,B 0,C 180,E1 -25345.354,E2 -25345.354} C_VEL
LIN {X 0,Y 207.264,Z 325.427,A -85,B 0,C 180,E1 -25346.616,E2 -25346.616} C_VEL
LIN {X 0,Y 214.457,Z 314.097,A -85,B 0,C 180,E1 -25347.551,E2 -25347.551} C_VEL
LIN {X 0,Y 217.22,Z 309.09,A -85,B 0,C 180,E1 -25347.869,E2 -25347.869} C_VEL
LIN {X 0,Y 218.095,Z 307.316,A -85,B 0,C 180,E1 -25348.394,E2 -25348.394} C_VEL
LIN {X 0,Y 212.089,Z 317.724,A -85,B 0,C 180,E1 -25349.36,E2 -25349.36} C_VEL
LIN {X 0,Y 204.485,Z 328.576,A -85,B 0,C 180,E1 -25350.674,E2 -25350.674} C_VEL
LIN {X 0,Y 196.169,Z 338.289,A -85,B 0,C 180,E1 -25352.241,E2 -25352.241} C_VEL
LIN {X 0,Y 187.445,Z 346.946,A -85,B 0,C 180,E1 -25354.14,E2 -25354.14} C_VEL
LIN {X 0,Y 178.928,Z 354.015,A -85,B 0,C 180,E1 -25356.258,E2 -25356.258} C_VEL
LIN {X 0,Y 171.481,Z 359.211,A -85,B 0,C 180,E1 -25358.354,E2 -25358.354} C_VEL
LIN {X 0,Y 163.579,Z 363.932,A -85,B 0,C 180,E1 -25360.948,E2 -25360.948} C_VEL
LIN {X 0,Y 155.102,Z 367.978,A -85,B 0,C 180,E1 -25364.223,E2 -25364.223} C_VEL
LIN {X 0,Y 150.137,Z 369.837,A -85,B 0,C 180,E1 -25366.463,E2 -25366.463} C_VEL
LIN {X 0,Y 142.494,Z 371.977,A -85,B 0,C 180,E1 -25370.555,E2 -25370.555} C_VEL
LIN {X 0,Y 137.113,Z 372.78,A -85,B 0,C 180,E1 -25374.115,E2 -25374.115} C_VEL
LIN {X 0,Y 133.504,Z 372.882,A -85,B 0,C 180,E1 -25376.981,E2 -25376.981} C_VEL
LIN {X 0,Y 130.308,Z 372.582,A -85,B 0,C 180,E1 -25379.999,E2 -25379.999} C_VEL
LIN {X 0,Y 126.807,Z 371.583,A -85,B 0,C 180,E1 -25383.947,E2 -25383.947} C_VEL
LIN {X 0,Y 123.077,Z 369.071,A -85,B 0,C 180,E1 -25389.863,E2 -25389.863} C_VEL
LIN {X 0,Y 120.884,Z 365.806,A -85,B 0,C 180,E1 -25395.165,E2 -25395.165} C_VEL
LIN {X 0,Y 119.697,Z 361.391,A -85,B 0,C 180,E1 -25400.626,E2 -25400.626} C_VEL
LIN {X 0,Y 119.521,Z 355.717,A -85,B 0,C 180,E1 -25406.167,E2 -25406.167} C_VEL
LIN {X 0,Y 120.066,Z 348.366,A -85,B 0,C 180,E1 -25411.789,E2 -25411.789} C_VEL
LIN {X 0,Y 120.949,Z 340.5,A -85,B 0,C 180,E1 -25416.554,E2 -25416.554} C_VEL
LIN {X 0,Y 122.351,Z 330.986,A -85,B 0,C 180,E1 -25421.19,E2 -25421.19} C_VEL
LIN {X 0,Y 124.025,Z 320.914,A -85,B 0,C 180,E1 -25425.097,E2 -25425.097} C_VEL
LIN {X 0,Y 126.075,Z 308.572,A -85,B 0,C 180,E1 -25428.885,E2 -25428.885} C_VEL
LIN {X 0,Y 127.951,Z 296.54,A -85,B 0,C 180,E1 -25431.72,E2 -25431.72} C_VEL
LIN {X 0,Y 129.735,Z 283.278,A -85,B 0,C 180,E1 -25434.097,E2 -25434.097} C_VEL
LIN {X 0,Y 131.141,Z 269.722,A -85,B 0,C 180,E1 -25435.822,E2 -25435.822} C_VEL
LIN {X 0,Y 133.243,Z 241.545,A -85,B 0,C 180,E1 -25438.115,E2 -25438.115} C_VEL
LIN {X 0,Y 135.442,Z 210.288,A -85,B 0,C 180,E1 -25440.457,E2 -25440.457} C_VEL
LIN {X 0,Y 126.235,Z 184.49,A -85,B 0,C 180,E1 -25443.979,E2 -25443.979} C_VEL
LIN {X 0,Y 122.021,Z 173.392,A -85,B 0,C 180,E1 -25445.714,E2 -25445.714} C_VEL
LIN {X 0,Y 122.02,Z 173.284,A -85,B 0,C 180,E1 -25449.781,E2 -25449.781} C_VEL
LIN {X 0,Y 122.242,Z 173.251,A -85,B 0,C 180,E1 -25456.703,E2 -25456.703} C_VEL
LIN {X 0,Y 122.444,Z 173.232,A -85,B 0,C 180,E1 -25460.083,E2 -25460.083} C_VEL
LIN {X 0,Y 122.605,Z 173.21,A -85,B 0,C 180,E1 -25466.713,E2 -25466.713} C_VEL
LIN {X 0,Y 123.042,Z 173.157,A -85,B 0,C 180,E1 -25469.999,E2 -25469.999} C_VEL
LIN {X 0,Y 122.445,Z 173.233,A -85,B 0,C 180,E1 -25476.591,E2 -25476.591} C_VEL
LIN {X 0,Y 122.445,Z 173.23,A -85,B 0,C 180,E1 -25479.914,E2 -25479.914} C_VEL
LIN {X 0,Y 122.26,Z 173.254,A -85,B 0,C 180,E1 -25483.292,E2 -25483.292} C_VEL
LIN {X 0,Y 122.042,Z 173.277,A -85,B 0,C 180,E1 -25490.212,E2 -25490.212} C_VEL
LIN {X 0,Y 121.979,Z 173.291,A -85,B 0,C 180,E1 -25493.784,E2 -25493.784} C_VEL
LIN {X 0,Y 121.926,Z 173.296,A -85,B 0,C 180,E1 -25500.163,E2 -25500.163} C_VEL
LIN {X 0,Y 121.934,Z 173.29,A -85,B 0,C 180,E1 -25506.205,E2 -25506.205} C_VEL
LIN {X 0,Y 121.94,Z 173.296,A -85,B 0,C 180,E1 -25511.476,E2 -25511.476} C_VEL
LIN {X 0,Y 121.939,Z 173.295,A -85,B 0,C 180,E1 -25518.524,E2 -25518.524} C_VEL
LIN {X 0,Y 121.974,Z 173.289,A -85,B 0,C 180,E1 -25524.819,E2 -25524.819} C_VEL
LIN {X 0,Y 121.939,Z 173.291,A -85,B 0,C 180,E1 -25529.826,E2 -25529.826} C_VEL
LIN {X 0,Y 121.981,Z 173.289,A -85,B 0,C 180,E1 -25536.216,E2 -25536.216} C_VEL
LIN {X 0,Y 122.047,Z 173.277,A -85,B 0,C 180,E1 -25539.789,E2 -25539.789} C_VEL
LIN {X 0,Y 122.261,Z 173.251,A -85,B 0,C 180,E1 -25546.708,E2 -25546.708} C_VEL
LIN {X 0,Y 122.445,Z 173.231,A -85,B 0,C 180,E1 -25550.086,E2 -25550.086} C_VEL
LIN {X 0,Y 122.604,Z 173.207,A -85,B 0,C 180,E1 -25556.715,E2 -25556.715} C_VEL
LIN {X 0,Y 123.042,Z 173.158,A -85,B 0,C 180,E1 -25560.001,E2 -25560.001} C_VEL
LIN {X 0,Y 122.455,Z 173.23,A -85,B 0,C 180,E1 -25566.592,E2 -25566.592} C_VEL
LIN {X 0,Y 122.455,Z 173.23,A -85,B 0,C 180,E1 -25569.916,E2 -25569.916} C_VEL
LIN {X 0,Y 122.261,Z 173.252,A -85,B 0,C 180,E1 -25573.294,E2 -25573.294} C_VEL
LIN {X 0,Y 122.044,Z 173.277,A -85,B 0,C 180,E1 -25580.214,E2 -25580.214} C_VEL
LIN {X 0,Y 121.981,Z 173.289,A -85,B 0,C 180,E1 -25583.786,E2 -25583.786} C_VEL
LIN {X 0,Y 121.929,Z 173.292,A -85,B 0,C 180,E1 -25590.165,E2 -25590.165} C_VEL
LIN {X 0,Y 121.913,Z 173.294,A -85,B 0,C 180,E1 -25596.192,E2 -25596.192} C_VEL
LIN {X 0,Y 121.909,Z 173.299,A -85,B 0,C 180,E1 -25601.46,E2 -25601.46} C_VEL
LIN {X 0,Y 121.997,Z 173.291,A -85,B 0,C 180,E1 -25607.925,E2 -25607.925} C_VEL
LIN {X 0,Y 126.851,Z 188.437,A -85,B 0,C 180,E1 -25610.18,E2 -25610.18} C_VEL
LIN {X 0,Y 132.235,Z 207.599,A -85,B 0,C 180,E1 -25612.631,E2 -25612.631} C_VEL
LIN {X 0,Y 134.234,Z 238.972,A -85,B 0,C 180,E1 -25615.523,E2 -25615.523} C_VEL
LIN {X 0,Y 131.195,Z 283.152,A -85,B 0,C 180,E1 -25619.016,E2 -25619.016} C_VEL
LIN {X 0,Y 129.872,Z 295.629,A -85,B 0,C 180,E1 -25620.545,E2 -25620.545} C_VEL
LIN {X 0,Y 128.147,Z 308.072,A -85,B 0,C 180,E1 -25622.659,E2 -25622.659} C_VEL
LIN {X 0,Y 126.013,Z 321.271,A -85,B 0,C 180,E1 -25625.714,E2 -25625.714} C_VEL
LIN {X 0,Y 123.98,Z 332.895,A -85,B 0,C 180,E1 -25629.251,E2 -25629.251} C_VEL
LIN {X 0,Y 122.437,Z 343.378,A -85,B 0,C 180,E1 -25633.323,E2 -25633.323} C_VEL
LIN {X 0,Y 121.431,Z 351.941,A -85,B 0,C 180,E1 -25637.466,E2 -25637.466} C_VEL
LIN {X 0,Y 120.88,Z 360.322,A -85,B 0,C 180,E1 -25642.558,E2 -25642.558} C_VEL
LIN {X 0,Y 120.843,Z 365.799,A -85,B 0,C 180,E1 -25646.667,E2 -25646.667} C_VEL
LIN {X 0,Y 120.926,Z 369.475,A -85,B 0,C 180,E1 -25650.001,E2 -25650.001} C_VEL
LIN {X 0,Y 120.628,Z 372.443,A -85,B 0,C 180,E1 -25653.341,E2 -25653.341} C_VEL
LIN {X 0,Y 120.345,Z 374.942,A -85,B 0,C 180,E1 -25656.879,E2 -25656.879} C_VEL
LIN {X 0,Y 120.88,Z 378.406,A -85,B 0,C 180,E1 -25663.449,E2 -25663.449} C_VEL
LIN {X 0,Y 123.074,Z 380.526,A -85,B 0,C 180,E1 -25670.038,E2 -25670.038} C_VEL
LIN {X 0,Y 127.221,Z 381.318,A -85,B 0,C 180,E1 -25676.229,E2 -25676.229} C_VEL
LIN {X 0,Y 132.91,Z 380.733,A -85,B 0,C 180,E1 -25681.924,E2 -25681.924} C_VEL
LIN {X 0,Y 139.992,Z 378.824,A -85,B 0,C 180,E1 -25687.046,E2 -25687.046} C_VEL
LIN {X 0,Y 148.473,Z 375.529,A -85,B 0,C 180,E1 -25691.507,E2 -25691.507} C_VEL
LIN {X 0,Y 157.889,Z 370.758,A -85,B 0,C 180,E1 -25695.415,E2 -25695.415} C_VEL
LIN {X 0,Y 161.129,Z 368.847,A -85,B 0,C 180,E1 -25696.561,E2 -25696.561} C_VEL
LIN {X 0,Y 164.713,Z 366.478,A -85,B 0,C 180,E1 -25697.99,E2 -25697.99} C_VEL
LIN {X 0,Y 173.699,Z 359.162,A -85,B 0,C 180,E1 -25702.584,E2 -25702.584} C_VEL
LIN {X 0,Y 177.259,Z 356.227,A -85,B 0,C 180,E1 -25703.769,E2 -25703.769} C_VEL
LIN {X 0,Y 178.59,Z 355.129,A -85,B 0,C 180,E1 -25704.077,E2 -25704.077} C_VEL
LIN {X 0,Y 188.178,Z 346.764,A -85,B 0,C 180,E1 -25705.929,E2 -25705.929} C_VEL
LIN {X 0,Y 197.238,Z 337.404,A -85,B 0,C 180,E1 -25707.351,E2 -25707.351} C_VEL
LIN {X 0,Y 203.876,Z 329.358,A -85,B 0,C 180,E1 -25708.261,E2 -25708.261} C_VEL
LIN {X 0,Y 204.375,Z 328.683,A -85,B 0,C 180,E1 -25708.576,E2 -25708.576} C_VEL
LIN {X 0,Y 196.37,Z 337.946,A -85,B 0,C 180,E1 -25709.929,E2 -25709.929} C_VEL
LIN {X 0,Y 188.025,Z 346.036,A -85,B 0,C 180,E1 -25711.537,E2 -25711.537} C_VEL
LIN {X 0,Y 178.231,Z 353.99,A -85,B 0,C 180,E1 -25713.686,E2 -25713.686} C_VEL
LIN {X 0,Y 169.249,Z 360.062,A -85,B 0,C 180,E1 -25716.001,E2 -25716.001} C_VEL
LIN {X 0,Y 161.5,Z 364.378,A -85,B 0,C 180,E1 -25718.29,E2 -25718.29} C_VEL
LIN {X 0,Y 153.038,Z 368.236,A -85,B 0,C 180,E1 -25721.248,E2 -25721.248} C_VEL
LIN {X 0,Y 146.145,Z 370.662,A -85,B 0,C 180,E1 -25724.113,E2 -25724.113} C_VEL
LIN {X 0,Y 137.893,Z 372.668,A -85,B 0,C 180,E1 -25728.236,E2 -25728.236} C_VEL
LIN {X 0,Y 133.504,Z 373.253,A -85,B 0,C 180,E1 -25730.912,E2 -25730.912} C_VEL
LIN {X 0,Y 126.835,Z 373.268,A -85,B 0,C 180,E1 -25735.875,E2 -25735.875} C_VEL
LIN {X 0,Y 122.57,Z 372.488,A -85,B 0,C 180,E1 -25739.999,E2 -25739.999} C_VEL
LIN {X 0,Y 119.69,Z 371.362,A -85,B 0,C 180,E1 -25743.411,E2 -25743.411} C_VEL
LIN {X 0,Y 117.394,Z 369.842,A -85,B 0,C 180,E1 -25746.875,E2 -25746.875} C_VEL
LIN {X 0,Y 114.895,Z 367.063,A -85,B 0,C 180,E1 -25751.839,E2 -25751.839} C_VEL
LIN {X 0,Y 113.032,Z 362.496,A -85,B 0,C 180,E1 -25758.111,E2 -25758.111} C_VEL
LIN {X 0,Y 112.446,Z 357.02,A -85,B 0,C 180,E1 -25763.968,E2 -25763.968} C_VEL
LIN {X 0,Y 112.792,Z 350.038,A -85,B 0,C 180,E1 -25769.898,E2 -25769.898} C_VEL
LIN {X 0,Y 113.65,Z 341.992,A -85,B 0,C 180,E1 -25775.289,E2 -25775.289} C_VEL
LIN {X 0,Y 114.978,Z 332.231,A -85,B 0,C 180,E1 -25780.498,E2 -25780.498} C_VEL
LIN {X 0,Y 116.559,Z 322.782,A -85,B 0,C 180,E1 -25784.536,E2 -25784.536} C_VEL
LIN {X 0,Y 118.465,Z 311.352,A -85,B 0,C 180,E1 -25788.386,E2 -25788.386} C_VEL
LIN {X 0,Y 120.526,Z 299.205,A -85,B 0,C 180,E1 -25791.585,E2 -25791.585} C_VEL
LIN {X 0,Y 122.306,Z 286.5,A -85,B 0,C 180,E1 -25794.117,E2 -25794.117} C_VEL
LIN {X 0,Y 123.917,Z 272.956,A -85,B 0,C 180,E1 -25796.09,E2 -25796.09} C_VEL
LIN {X 0,Y 125.277,Z 256.24,A -85,B 0,C 180,E1 -25797.67,E2 -25797.67} C_VEL
LIN {X 0,Y 128.528,Z 211.448,A -85,B 0,C 180,E1 -25801.243,E2 -25801.243} C_VEL
LIN {X 0,Y 119.931,Z 187.272,A -85,B 0,C 180,E1 -25804.774,E2 -25804.774} C_VEL
LIN {X 0,Y 115.018,Z 174.317,A -85,B 0,C 180,E1 -25806.957,E2 -25806.957} C_VEL
LIN {X 0,Y 114.988,Z 174.161,A -85,B 0,C 180,E1 -25812.205,E2 -25812.205} C_VEL
LIN {X 0,Y 115.262,Z 174.122,A -85,B 0,C 180,E1 -25817.307,E2 -25817.307} C_VEL
LIN {X 0,Y 115.386,Z 174.109,A -85,B 0,C 180,E1 -25823.002,E2 -25823.002} C_VEL
LIN {X 0,Y 115.994,Z 174.035,A -85,B 0,C 180,E1 -25829.999,E2 -25829.999} C_VEL
LIN {X 0,Y 115.387,Z 174.112,A -85,B 0,C 180,E1 -25836.996,E2 -25836.996} C_VEL
LIN {X 0,Y 115.282,Z 174.121,A -85,B 0,C 180,E1 -25842.737,E2 -25842.737} C_VEL
LIN {X 0,Y 115.01,Z 174.157,A -85,B 0,C 180,E1 -25847.789,E2 -25847.789} C_VEL
LIN {X 0,Y 114.944,Z 174.167,A -85,B 0,C 180,E1 -25853.492,E2 -25853.492} C_VEL
LIN {X 0,Y 114.861,Z 174.177,A -85,B 0,C 180,E1 -25861.064,E2 -25861.064} C_VEL
LIN {X 0,Y 114.845,Z 174.175,A -85,B 0,C 180,E1 -25867.729,E2 -25867.729} C_VEL
LIN {X 0,Y 114.863,Z 174.174,A -85,B 0,C 180,E1 -25872.759,E2 -25872.759} C_VEL
LIN {X 0,Y 114.867,Z 174.177,A -85,B 0,C 180,E1 -25877.701,E2 -25877.701} C_VEL
LIN {X 0,Y 114.852,Z 174.171,A -85,B 0,C 180,E1 -25882.699,E2 -25882.699} C_VEL
LIN {X 0,Y 114.867,Z 174.175,A -85,B 0,C 180,E1 -25888.931,E2 -25888.931} C_VEL
LIN {X 0,Y 114.944,Z 174.166,A -85,B 0,C 180,E1 -25896.508,E2 -25896.508} C_VEL
LIN {X 0,Y 115.015,Z 174.157,A -85,B 0,C 180,E1 -25902.212,E2 -25902.212} C_VEL
LIN {X 0,Y 115.282,Z 174.119,A -85,B 0,C 180,E1 -25907.263,E2 -25907.263} C_VEL
LIN {X 0,Y 115.387,Z 174.111,A -85,B 0,C 180,E1 -25913.004,E2 -25913.004} C_VEL
LIN {X 0,Y 115.994,Z 174.036,A -85,B 0,C 180,E1 -25920.001,E2 -25920.001} C_VEL
LIN {X 0,Y 115.396,Z 174.111,A -85,B 0,C 180,E1 -25926.998,E2 -25926.998} C_VEL
LIN {X 0,Y 115.392,Z 174.108,A -85,B 0,C 180,E1 -25930.529,E2 -25930.529} C_VEL
LIN {X 0,Y 115.145,Z 174.139,A -85,B 0,C 180,E1 -25934.133,E2 -25934.133} C_VEL
LIN {X 0,Y 114.98,Z 174.157,A -85,B 0,C 180,E1 -25941.516,E2 -25941.516} C_VEL
LIN {X 0,Y 114.866,Z 174.176,A -85,B 0,C 180,E1 -25945.361,E2 -25945.361} C_VEL
LIN {X 0,Y 114.863,Z 174.175,A -85,B 0,C 180,E1 -25951.066,E2 -25951.066} C_VEL
LIN {X 0,Y 114.811,Z 174.177,A -85,B 0,C 180,E1 -25957.746,E2 -25957.746} C_VEL
LIN {X 0,Y 114.842,Z 174.173,A -85,B 0,C 180,E1 -25964.801,E2 -25964.801} C_VEL
LIN {X 0,Y 114.926,Z 174.352,A -85,B 0,C 180,E1 -25966.742,E2 -25966.742} C_VEL
LIN {X 0,Y 118.802,Z 185.455,A -85,B 0,C 180,E1 -25968.563,E2 -25968.563} C_VEL
LIN {X 0,Y 125.43,Z 208.625,A -85,B 0,C 180,E1 -25971.782,E2 -25971.782} C_VEL
LIN {X 0,Y 127.386,Z 238.997,A -85,B 0,C 180,E1 -25974.738,E2 -25974.738} C_VEL
LIN {X 0,Y 124.203,Z 283.187,A -85,B 0,C 180,E1 -25978.468,E2 -25978.468} C_VEL
LIN {X 0,Y 122.773,Z 296.12,A -85,B 0,C 180,E1 -25980.18,E2 -25980.18} C_VEL
LIN {X 0,Y 121.067,Z 307.877,A -85,B 0,C 180,E1 -25982.33,E2 -25982.33} C_VEL
LIN {X 0,Y 118.908,Z 321.038,A -85,B 0,C 180,E1 -25985.562,E2 -25985.562} C_VEL
LIN {X 0,Y 116.833,Z 332.6,A -85,B 0,C 180,E1 -25989.306,E2 -25989.306} C_VEL
LIN {X 0,Y 115.435,Z 342.099,A -85,B 0,C 180,E1 -25993.192,E2 -25993.192} C_VEL
LIN {X 0,Y 114.451,Z 350.812,A -85,B 0,C 180,E1 -25997.59,E2 -25997.59} C_VEL
LIN {X 0,Y 113.908,Z 357.987,A -85,B 0,C 180,E1 -26002.044,E2 -26002.044} C_VEL
LIN {X 0,Y 113.917,Z 363.805,A -85,B 0,C 180,E1 -26006.464,E2 -26006.464} C_VEL
LIN {X 0,Y 113.992,Z 367.681,A -85,B 0,C 180,E1 -26010.001,E2 -26010.001} C_VEL
LIN {X 0,Y 113.993,Z 369.337,A -85,B 0,C 180,E1 -26011.768,E2 -26011.768} C_VEL
LIN {X 0,Y 113.45,Z 373.686,A -85,B 0,C 180,E1 -26017.611,E2 -26017.611} C_VEL
LIN {X 0,Y 114.066,Z 377.259,A -85,B 0,C 180,E1 -26024.269,E2 -26024.269} C_VEL
LIN {X 0,Y 116.475,Z 379.637,A -85,B 0,C 180,E1 -26031.226,E2 -26031.226} C_VEL
LIN {X 0,Y 120.9,Z 380.711,A -85,B 0,C 180,E1 -26037.715,E2 -26037.715} C_VEL
LIN {X 0,Y 126.93,Z 380.468,A -85,B 0,C 180,E1 -26043.622,E2 -26043.622} C_VEL
LIN {X 0,Y 134.409,Z 378.921,A -85,B 0,C 180,E1 -26048.864,E2 -26048.864} C_VEL
LIN {X 0,Y 143.254,Z 376.008,A -85,B 0,C 180,E1 -26053.382,E2 -26053.382} C_VEL
LIN {X 0,Y 153.034,Z 371.625,A -85,B 0,C 180,E1 -26057.291,E2 -26057.291} C_VEL
LIN {X 0,Y 161.008,Z 367.322,A -85,B 0,C 180,E1 -26059.808,E2 -26059.808} C_VEL
LIN {X 0,Y 170.832,Z 361.005,A -85,B 0,C 180,E1 -26062.368,E2 -26062.368} C_VEL
LIN {X 0,Y 178.59,Z 355.129,A -85,B 0,C 180,E1 -26064.077,E2 -26064.077} C_VEL
LIN {X 0,Y 182.13,Z 352.152,A -85,B 0,C 180,E1 -26064.965,E2 -26064.965} C_VEL
LIN {X 0,Y 185.184,Z 349.325,A -85,B 0,C 180,E1 -26066.042,E2 -26066.042} C_VEL
LIN {X 0,Y 188.299,Z 346.138,A -85,B 0,C 180,E1 -26067.614,E2 -26067.614} C_VEL
LIN {X 0,Y 189.762,Z 344.573,A -85,B 0,C 180,E1 -26068.667,E2 -26068.667} C_VEL
LIN {X 0,Y 189.914,Z 344.416,A -85,B 0,C 180,E1 -26068.795,E2 -26068.795} C_VEL
LIN {X 0,Y 181.439,Z 351.512,A -85,B 0,C 180,E1 -26070.404,E2 -26070.404} C_VEL
LIN {X 0,Y 173.142,Z 357.355,A -85,B 0,C 180,E1 -26072.171,E2 -26072.171} C_VEL
LIN {X 0,Y 163.394,Z 363.079,A -85,B 0,C 180,E1 -26074.592,E2 -26074.592} C_VEL
LIN {X 0,Y 154.399,Z 367.342,A -85,B 0,C 180,E1 -26077.237,E2 -26077.237} C_VEL
LIN {X 0,Y 145.763,Z 370.5,A -85,B 0,C 180,E1 -26080.274,E2 -26080.274} C_VEL
LIN {X 0,Y 139.828,Z 372.124,A -85,B 0,C 180,E1 -26082.744,E2 -26082.744} C_VEL
LIN {X 0,Y 130.359,Z 373.733,A -85,B 0,C 180,E1 -26087.545,E2 -26087.545} C_VEL
LIN {X 0,Y 125.881,Z 373.923,A -85,B 0,C 180,E1 -26090.357,E2 -26090.357} C_VEL
LIN {X 0,Y 119.954,Z 373.477,A -85,B 0,C 180,E1 -26094.895,E2 -26094.895} C_VEL
LIN {X 0,Y 114.859,Z 372.065,A -85,B 0,C 180,E1 -26099.999,E2 -26099.999} C_VEL
LIN {X 0,Y 112.058,Z 370.588,A -85,B 0,C 180,E1 -26103.594,E2 -26103.594} C_VEL
LIN {X 0,Y 108.763,Z 367.589,A -85,B 0,C 180,E1 -26109.295,E2 -26109.295} C_VEL
LIN {X 0,Y 106.587,Z 363.506,A -85,B 0,C 180,E1 -26115.291,E2 -26115.291} C_VEL
LIN {X 0,Y 105.517,Z 357.585,A -85,B 0,C 180,E1 -26122.172,E2 -26122.172} C_VEL
LIN {X 0,Y 105.544,Z 351.566,A -85,B 0,C 180,E1 -26127.781,E2 -26127.781} C_VEL
LIN {X 0,Y 106.233,Z 344.538,A -85,B 0,C 180,E1 -26133.077,E2 -26133.077} C_VEL
LIN {X 0,Y 107.266,Z 336.234,A -85,B 0,C 180,E1 -26138.163,E2 -26138.163} C_VEL
LIN {X 0,Y 108.903,Z 325.739,A -85,B 0,C 180,E1 -26143.287,E2 -26143.287} C_VEL
LIN {X 0,Y 110.702,Z 315.233,A -85,B 0,C 180,E1 -26147.359,E2 -26147.359} C_VEL
LIN {X 0,Y 112.617,Z 304.204,A -85,B 0,C 180,E1 -26150.758,E2 -26150.758} C_VEL
LIN {X 0,Y 114.559,Z 292.124,A -85,B 0,C 180,E1 -26153.627,E2 -26153.627} C_VEL
LIN {X 0,Y 116.245,Z 279.686,A -85,B 0,C 180,E1 -26155.843,E2 -26155.843} C_VEL
LIN {X 0,Y 117.557,Z 266.083,A -85,B 0,C 180,E1 -26157.556,E2 -26157.556} C_VEL
LIN {X 0,Y 121.708,Z 212.986,A -85,B 0,C 180,E1 -26162.064,E2 -26162.064} C_VEL
LIN {X 0,Y 113.691,Z 190.213,A -85,B 0,C 180,E1 -26165.606,E2 -26165.606} C_VEL
LIN {X 0,Y 107.936,Z 175.04,A -85,B 0,C 180,E1 -26168.388,E2 -26168.388} C_VEL
LIN {X 0,Y 108.182,Z 175.003,A -85,B 0,C 180,E1 -26177.018,E2 -26177.018} C_VEL
LIN {X 0,Y 108.325,Z 174.99,A -85,B 0,C 180,E1 -26182.543,E2 -26182.543} C_VEL
LIN {X 0,Y 108.944,Z 174.914,A -85,B 0,C 180,E1 -26189.999,E2 -26189.999} C_VEL
LIN {X 0,Y 108.327,Z 174.991,A -85,B 0,C 180,E1 -26197.454,E2 -26197.454} C_VEL
LIN {X 0,Y 108.197,Z 175.005,A -85,B 0,C 180,E1 -26203.015,E2 -26203.015} C_VEL
LIN {X 0,Y 107.903,Z 175.037,A -85,B 0,C 180,E1 -26209.004,E2 -26209.004} C_VEL
LIN {X 0,Y 107.853,Z 175.051,A -85,B 0,C 180,E1 -26214.182,E2 -26214.182} C_VEL
LIN {X 0,Y 107.793,Z 175.059,A -85,B 0,C 180,E1 -26222.052,E2 -26222.052} C_VEL
LIN {X 0,Y 107.752,Z 175.062,A -85,B 0,C 180,E1 -26228.495,E2 -26228.495} C_VEL
LIN {X 0,Y 107.766,Z 175.057,A -85,B 0,C 180,E1 -26235.836,E2 -26235.836} C_VEL
LIN {X 0,Y 107.752,Z 175.058,A -85,B 0,C 180,E1 -26241.505,E2 -26241.505} C_VEL
LIN {X 0,Y 107.809,Z 175.054,A -85,B 0,C 180,E1 -26248.568,E2 -26248.568} C_VEL
LIN {X 0,Y 107.908,Z 175.042,A -85,B 0,C 180,E1 -26256.999,E2 -26256.999} C_VEL
LIN {X 0,Y 108.037,Z 175.027,A -85,B 0,C 180,E1 -26264.919,E2 -26264.919} C_VEL
LIN {X 0,Y 108.286,Z 174.991,A -85,B 0,C 180,E1 -26268.774,E2 -26268.774} C_VEL
LIN {X 0,Y 108.455,Z 174.968,A -85,B 0,C 180,E1 -26276.286,E2 -26276.286} C_VEL
LIN {X 0,Y 108.944,Z 174.914,A -85,B 0,C 180,E1 -26280.001,E2 -26280.001} C_VEL
LIN {X 0,Y 108.339,Z 174.989,A -85,B 0,C 180,E1 -26287.456,E2 -26287.456} C_VEL
LIN {X 0,Y 108.202,Z 175.001,A -85,B 0,C 180,E1 -26293.027,E2 -26293.027} C_VEL
LIN {X 0,Y 107.904,Z 175.04,A -85,B 0,C 180,E1 -26299.007,E2 -26299.007} C_VEL
LIN {X 0,Y 107.855,Z 175.05,A -85,B 0,C 180,E1 -26304.184,E2 -26304.184} C_VEL
LIN {X 0,Y 107.791,Z 175.058,A -85,B 0,C 180,E1 -26312.051,E2 -26312.051} C_VEL
LIN {X 0,Y 107.719,Z 175.063,A -85,B 0,C 180,E1 -26318.473,E2 -26318.473} C_VEL
LIN {X 0,Y 107.809,Z 175.05,A -85,B 0,C 180,E1 -26325.269,E2 -26325.269} C_VEL
LIN {X 0,Y 110.203,Z 181.279,A -85,B 0,C 180,E1 -26326.506,E2 -26326.506} C_VEL
LIN {X 0,Y 114.44,Z 194.709,A -85,B 0,C 180,E1 -26328.694,E2 -26328.694} C_VEL
LIN {X 0,Y 118.775,Z 210.542,A -85,B 0,C 180,E1 -26330.979,E2 -26330.979} C_VEL
LIN {X 0,Y 120.449,Z 239.863,A -85,B 0,C 180,E1 -26333.994,E2 -26333.994} C_VEL
LIN {X 0,Y 117.33,Z 282.194,A -85,B 0,C 180,E1 -26337.761,E2 -26337.761} C_VEL
LIN {X 0,Y 115.738,Z 296.025,A -85,B 0,C 180,E1 -26339.686,E2 -26339.686} C_VEL
LIN {X 0,Y 114.003,Z 307.691,A -85,B 0,C 180,E1 -26341.963,E2 -26341.963} C_VEL
LIN {X 0,Y 111.779,Z 320.785,A -85,B 0,C 180,E1 -26345.385,E2 -26345.385} C_VEL
LIN {X 0,Y 109.909,Z 331.181,A -85,B 0,C 180,E1 -26348.921,E2 -26348.921} C_VEL
LIN {X 0,Y 108.463,Z 340.775,A -85,B 0,C 180,E1 -26353.049,E2 -26353.049} C_VEL
LIN {X 0,Y 107.487,Z 349.567,A -85,B 0,C 180,E1 -26357.733,E2 -26357.733} C_VEL
LIN {X 0,Y 106.993,Z 358.107,A -85,B 0,C 180,E1 -26363.401,E2 -26363.401} C_VEL
LIN {X 0,Y 107.033,Z 363.796,A -85,B 0,C 180,E1 -26368.12,E2 -26368.12} C_VEL
LIN {X 0,Y 107.107,Z 367.534,A -85,B 0,C 180,E1 -26371.881,E2 -26371.881} C_VEL
LIN {X 0,Y 106.576,Z 372.353,A -85,B 0,C 180,E1 -26378.438,E2 -26378.438} C_VEL
LIN {X 0,Y 107.306,Z 375.954,A -85,B 0,C 180,E1 -26385.189,E2 -26385.189} C_VEL
LIN {X 0,Y 109.931,Z 378.666,A -85,B 0,C 180,E1 -26392.558,E2 -26392.558} C_VEL
LIN {X 0,Y 114.671,Z 380.056,A -85,B 0,C 180,E1 -26399.362,E2 -26399.362} C_VEL
LIN {X 0,Y 121.068,Z 380.139,A -85,B 0,C 180,E1 -26405.487,E2 -26405.487} C_VEL
LIN {X 0,Y 128.96,Z 378.918,A -85,B 0,C 180,E1 -26410.843,E2 -26410.843} C_VEL
LIN {X 0,Y 138.19,Z 376.378,A -85,B 0,C 180,E1 -26415.4,E2 -26415.4} C_VEL
LIN {X 0,Y 148.354,Z 372.478,A -85,B 0,C 180,E1 -26419.287,E2 -26419.287} C_VEL
LIN {X 0,Y 156.574,Z 368.507,A -85,B 0,C 180,E1 -26421.769,E2 -26421.769} C_VEL
LIN {X 0,Y 165.194,Z 363.568,A -85,B 0,C 180,E1 -26423.935,E2 -26423.935} C_VEL
LIN {X 0,Y 175.75,Z 356.45,A -85,B 0,C 180,E1 -26426.137,E2 -26426.137} C_VEL
LIN {X 0,Y 185.59,Z 348.431,A -85,B 0,C 180,E1 -26427.895,E2 -26427.895} C_VEL
LIN {X 0,Y 189.572,Z 344.771,A -85,B 0,C 180,E1 -26428.506,E2 -26428.506} C_VEL
LIN {X 0,Y 189.762,Z 344.573,A -85,B 0,C 180,E1 -26428.667,E2 -26428.667} C_VEL
LIN {X 0,Y 189.646,Z 344.647,A -85,B 0,C 180,E1 -26429.127,E2 -26429.127} C_VEL
LIN {X 0,Y 188.142,Z 345.954,A -85,B 0,C 180,E1 -26429.736,E2 -26429.736} C_VEL
LIN {X 0,Y 184.642,Z 348.95,A -85,B 0,C 180,E1 -26430.229,E2 -26430.229} C_VEL
LIN {X 0,Y 181.722,Z 351.286,A -85,B 0,C 180,E1 -26430.375,E2 -26430.375} C_VEL
LIN {X 0,Y 171.195,Z 358.66,A -85,B 0,C 180,E1 -26430.508,E2 -26430.508} C_VEL
LIN {X 0,Y 166.5,Z 361.432,A -85,B 0,C 180,E1 -26430.99,E2 -26430.99} C_VEL
LIN {X 0,Y 165.025,Z 362.212,A -85,B 0,C 180,E1 -26431.278,E2 -26431.278} C_VEL
LIN {X 0,Y 156.635,Z 366.28,A -85,B 0,C 180,E1 -26433.34,E2 -26433.34} C_VEL
LIN {X 0,Y 145.378,Z 370.531,A -85,B 0,C 180,E1 -26436.712,E2 -26436.712} C_VEL
LIN {X 0,Y 138.492,Z 372.415,A -85,B 0,C 180,E1 -26439.192,E2 -26439.192} C_VEL
LIN {X 0,Y 132.953,Z 373.511,A -85,B 0,C 180,E1 -26441.507,E2 -26441.507} C_VEL
LIN {X 0,Y 127.722,Z 374.195,A -85,B 0,C 180,E1 -26444.029,E2 -26444.029} C_VEL
LIN {X 0,Y 122.723,Z 374.451,A -85,B 0,C 180,E1 -26446.795,E2 -26446.795} C_VEL
LIN {X 0,Y 114.097,Z 373.686,A -85,B 0,C 180,E1 -26452.922,E2 -26452.922} C_VEL
LIN {X 0,Y 110.381,Z 372.715,A -85,B 0,C 180,E1 -26456.348,E2 -26456.348} C_VEL
LIN {X 0,Y 105.498,Z 370.316,A -85,B 0,C 180,E1 -26462.165,E2 -26462.165} C_VEL
LIN {X 0,Y 102.114,Z 367.195,A -85,B 0,C 180,E1 -26467.91,E2 -26467.91} C_VEL
LIN {X 0,Y 99.746,Z 362.915,A -85,B 0,C 180,E1 -26474.275,E2 -26474.275} C_VEL
LIN {X 0,Y 98.582,Z 357.399,A -85,B 0,C 180,E1 -26480.881,E2 -26480.881} C_VEL
LIN {X 0,Y 98.564,Z 350.453,A -85,B 0,C 180,E1 -26487.61,E2 -26487.61} C_VEL
LIN {X 0,Y 99.316,Z 342.763,A -85,B 0,C 180,E1 -26493.577,E2 -26493.577} C_VEL
LIN {X 0,Y 100.416,Z 333.958,A -85,B 0,C 180,E1 -26499.041,E2 -26499.041} C_VEL
LIN {X 0,Y 102.11,Z 323.627,A -85,B 0,C 180,E1 -26504.164,E2 -26504.164} C_VEL
LIN {X 0,Y 104.14,Z 312.005,A -85,B 0,C 180,E1 -26508.656,E2 -26508.656} C_VEL
LIN {X 0,Y 106.384,Z 299.318,A -85,B 0,C 180,E1 -26512.441,E2 -26512.441} C_VEL
LIN {X 0,Y 108.291,Z 286.445,A -85,B 0,C 180,E1 -26515.304,E2 -26515.304} C_VEL
LIN {X 0,Y 110.033,Z 272.879,A -85,B 0,C 180,E1 -26517.488,E2 -26517.488} C_VEL
LIN {X 0,Y 111.687,Z 253.388,A -85,B 0,C 180,E1 -26519.499,E2 -26519.499} C_VEL
LIN {X 0,Y 114.767,Z 214.103,A -85,B 0,C 180,E1 -26523.03,E2 -26523.03} C_VEL
LIN {X 0,Y 107.48,Z 193.26,A -85,B 0,C 180,E1 -26526.441,E2 -26526.441} C_VEL
LIN {X 0,Y 100.852,Z 175.921,A -85,B 0,C 180,E1 -26529.873,E2 -26529.873} C_VEL
LIN {X 0,Y 101.172,Z 175.879,A -85,B 0,C 180,E1 -26537.97,E2 -26537.97} C_VEL
LIN {X 0,Y 101.262,Z 175.87,A -85,B 0,C 180,E1 -26542.02,E2 -26542.02} C_VEL
LIN {X 0,Y 101.868,Z 175.795,A -85,B 0,C 180,E1 -26549.999,E2 -26549.999} C_VEL
LIN {X 0,Y 101.266,Z 175.871,A -85,B 0,C 180,E1 -26557.977,E2 -26557.977} C_VEL
LIN {X 0,Y 101.122,Z 175.887,A -85,B 0,C 180,E1 -26563.351,E2 -26563.351} C_VEL
LIN {X 0,Y 100.814,Z 175.921,A -85,B 0,C 180,E1 -26570.398,E2 -26570.398} C_VEL
LIN {X 0,Y 100.771,Z 175.931,A -85,B 0,C 180,E1 -26574.958,E2 -26574.958} C_VEL
LIN {X 0,Y 100.702,Z 175.94,A -85,B 0,C 180,E1 -26583.128,E2 -26583.128} C_VEL
LIN {X 0,Y 100.699,Z 175.942,A -85,B 0,C 180,E1 -26589.853,E2 -26589.853} C_VEL
LIN {X 0,Y 100.732,Z 175.932,A -85,B 0,C 180,E1 -26595.76,E2 -26595.76} C_VEL
LIN {X 0,Y 100.693,Z 175.939,A -85,B 0,C 180,E1 -26601.087,E2 -26601.087} C_VEL
LIN {X 0,Y 100.705,Z 175.941,A -85,B 0,C 180,E1 -26606.87,E2 -26606.87} C_VEL
LIN {X 0,Y 100.783,Z 175.932,A -85,B 0,C 180,E1 -26615.268,E2 -26615.268} C_VEL
LIN {X 0,Y 100.816,Z 175.92,A -85,B 0,C 180,E1 -26619.603,E2 -26619.603} C_VEL
LIN {X 0,Y 101.186,Z 175.874,A -85,B 0,C 180,E1 -26627.975,E2 -26627.975} C_VEL
LIN {X 0,Y 101.265,Z 175.871,A -85,B 0,C 180,E1 -26632.023,E2 -26632.023} C_VEL
LIN {X 0,Y 101.868,Z 175.796,A -85,B 0,C 180,E1 -26640.001,E2 -26640.001} C_VEL
LIN {X 0,Y 101.278,Z 175.869,A -85,B 0,C 180,E1 -26647.979,E2 -26647.979} C_VEL
LIN {X 0,Y 101.113,Z 175.885,A -85,B 0,C 180,E1 -26653.328,E2 -26653.328} C_VEL
LIN {X 0,Y 100.816,Z 175.92,A -85,B 0,C 180,E1 -26660.401,E2 -26660.401} C_VEL
LIN {X 0,Y 100.774,Z 175.932,A -85,B 0,C 180,E1 -26664.96,E2 -26664.96} C_VEL
LIN {X 0,Y 100.698,Z 175.941,A -85,B 0,C 180,E1 -26673.125,E2 -26673.125} C_VEL
LIN {X 0,Y 100.669,Z 175.944,A -85,B 0,C 180,E1 -26679.833,E2 -26679.833} C_VEL
LIN {X 0,Y 100.716,Z 175.935,A -85,B 0,C 180,E1 -26683.788,E2 -26683.788} C_VEL
LIN {X 0,Y 105.351,Z 188.119,A -85,B 0,C 180,E1 -26686.263,E2 -26686.263} C_VEL
LIN {X 0,Y 112.077,Z 211.919,A -85,B 0,C 180,E1 -26690.017,E2 -26690.017} C_VEL
LIN {X 0,Y 113.59,Z 240.272,A -85,B 0,C 180,E1 -26693.126,E2 -26693.126} C_VEL
LIN {X 0,Y 110.344,Z 282.198,A -85,B 0,C 180,E1 -26697.088,E2 -26697.088} C_VEL
LIN {X 0,Y 108.732,Z 295.834,A -85,B 0,C 180,E1 -26699.134,E2 -26699.134} C_VEL
LIN {X 0,Y 106.608,Z 309.097,A -85,B 0,C 180,E1 -26701.986,E2 -26701.986} C_VEL
LIN {X 0,Y 104.687,Z 320.311,A -85,B 0,C 180,E1 -26705.193,E2 -26705.193} C_VEL
LIN {X 0,Y 102.814,Z 330.644,A -85,B 0,C 180,E1 -26708.971,E2 -26708.971} C_VEL
LIN {X 0,Y 101.279,Z 341.203,A -85,B 0,C 180,E1 -26713.886,E2 -26713.886} C_VEL
LIN {X 0,Y 100.303,Z 350.234,A -85,B 0,C 180,E1 -26719.165,E2 -26719.165} C_VEL
LIN {X 0,Y 100.064,Z 358.194,A -85,B 0,C 180,E1 -26724.965,E2 -26724.965} C_VEL
LIN {X 0,Y 100.192,Z 363.766,A -85,B 0,C 180,E1 -26730.001,E2 -26730.001} C_VEL
LIN {X 0,Y 100.258,Z 365.619,A -85,B 0,C 180,E1 -26732.01,E2 -26732.01} C_VEL
LIN {X 0,Y 99.738,Z 370.1,A -85,B 0,C 180,E1 -26738.103,E2 -26738.103} C_VEL
LIN {X 0,Y 100.565,Z 374.604,A -85,B 0,C 180,E1 -26746.234,E2 -26746.234} C_VEL
LIN {X 0,Y 103.475,Z 377.598,A -85,B 0,C 180,E1 -26754.051,E2 -26754.051} C_VEL
LIN {X 0,Y 108.566,Z 379.283,A -85,B 0,C 180,E1 -26761.192,E2 -26761.192} C_VEL
LIN {X 0,Y 116.131,Z 379.666,A -85,B 0,C 180,E1 -26768.117,E2 -26768.117} C_VEL
LIN {X 0,Y 123.691,Z 378.837,A -85,B 0,C 180,E1 -26772.988,E2 -26772.988} C_VEL
LIN {X 0,Y 133.319,Z 376.71,A -85,B 0,C 180,E1 -26777.564,E2 -26777.564} C_VEL
LIN {X 0,Y 143.848,Z 373.2,A -85,B 0,C 180,E1 -26781.419,E2 -26781.419} C_VEL
LIN {X 0,Y 155.221,Z 368.197,A -85,B 0,C 180,E1 -26784.588,E2 -26784.588} C_VEL
LIN {X 0,Y 164.206,Z 363.362,A -85,B 0,C 180,E1 -26786.575,E2 -26786.575} C_VEL
LIN {X 0,Y 175.063,Z 356.305,A -85,B 0,C 180,E1 -26788.595,E2 -26788.595} C_VEL
LIN {X 0,Y 174.77,Z 356.429,A -85,B 0,C 180,E1 -26789.187,E2 -26789.187} C_VEL
LIN {X 0,Y 165.025,Z 362.212,A -85,B 0,C 180,E1 -26791.278,E2 -26791.278} C_VEL
LIN {X 0,Y 160.209,Z 364.675,A -85,B 0,C 180,E1 -26792.146,E2 -26792.146} C_VEL
LIN {X 0,Y 151.433,Z 368.463,A -85,B 0,C 180,E1 -26793.157,E2 -26793.157} C_VEL
LIN {X 0,Y 144.317,Z 370.928,A -85,B 0,C 180,E1 -26794.069,E2 -26794.069} C_VEL
LIN {X 0,Y 139.285,Z 372.327,A -85,B 0,C 180,E1 -26795.141,E2 -26795.141} C_VEL
LIN {X 0,Y 137.751,Z 372.695,A -85,B 0,C 180,E1 -26795.614,E2 -26795.614} C_VEL
LIN {X 0,Y 127.538,Z 374.479,A -85,B 0,C 180,E1 -26799.522,E2 -26799.522} C_VEL
LIN {X 0,Y 120.245,Z 374.974,A -85,B 0,C 180,E1 -26803.007,E2 -26803.007} C_VEL
LIN {X 0,Y 115.23,Z 374.823,A -85,B 0,C 180,E1 -26805.878,E2 -26805.878} C_VEL
LIN {X 0,Y 106.424,Z 373.326,A -85,B 0,C 180,E1 -26812.409,E2 -26812.409} C_VEL
LIN {X 0,Y 102.695,Z 371.99,A -85,B 0,C 180,E1 -26816.074,E2 -26816.074} C_VEL
LIN {X 0,Y 98.424,Z 369.49,A -85,B 0,C 180,E1 -26821.416,E2 -26821.416} C_VEL
LIN {X 0,Y 94.531,Z 365.338,A -85,B 0,C 180,E1 -26828.55,E2 -26828.55} C_VEL
